
	    #sw_NumberOfFailsAux.%X0 := NOT #ix_PowerSupplyOk_1;            //  Power supply 1 state
	    #sw_NumberOfFailsAux.%X1 := NOT #ix_PowerSupplyOk_2;            //  Power supply 2 state
	    #sw_NumberOfFailsAux.%X2 := NOT #ix_PowerSupplyOk_3;            //  Power supply 3 state
	    #sw_NumberOfFailsAux.%X3 := NOT #ix_PowerSupplyOk_4;            //  Power supply 4 state
	    #sw_NumberOfFailsAux.%X4 := NOT #ix_PowerSupplyOk_5;            //  Power supply 5 state
	    #sw_NumberOfFailsAux.%X5 := NOT #ix_PowerSupplyOk_6;            //  Power supply 6 state
	    #sw_NumberOfFailsAux.%X6 := NOT #ix_PowerSupplyOk_7;            //  Power supply 7 state
	    #sw_NumberOfFailsAux.%X7 := NOT #ix_PowerSupplyOk_8;            //  Power supply 8 state
	    #sw_NumberOfFailsAux.%X8 := NOT #ix_PowerSupplyOk_9;            //  Power supply 9 state
	    #sw_NumberOfFailsAux.%X9 := NOT #ix_PowerSupplyOk_10;           //  Power supply 10 state

	    #si_NumberOfFails := BITSUM(#sw_NumberOfFailsAux);

	END_REGION

	REGION 2 - Reset

	    IF #iqUDT_EquipmentControl.Command.Reset
	    THEN

	        #sUDT_HMIStatus.Specific.Fail_PowerSupply_1 := FALSE;      //  Power supply fault state
	        #sUDT_HMIStatus.Specific.Fail_PowerSupply_2 := FALSE;      //  Power supply fault state
	        #sUDT_HMIStatus.Specific.Fail_PowerSupply_3 := FALSE;      //  Power supply fault state
	        #sUDT_HMIStatus.Specific.Fail_PowerSupply_4 := FALSE;      //  Power supply fault state
	        #sUDT_HMIStatus.Specific.Fail_PowerSupply_5 := FALSE;      //  Power supply fault state
	        #sUDT_HMIStatus.Specific.Fail_PowerSupply_6 := FALSE;      //  Power supply fault state
	        #sUDT_HMIStatus.Specific.Fail_PowerSupply_7 := FALSE;      //  Power supply fault state
	        #sUDT_HMIStatus.Specific.Fail_PowerSupply_8 := FALSE;      //  Power supply fault state
	        #sUDT_HMIStatus.Specific.Fail_PowerSupply_9 := FALSE;      //  Power supply fault state
	        #sUDT_HMIStatus.Specific.Fail_PowerSupply_10 := FALSE;     //  Power supply fault state

	        #sUDT_HMIStatus.Specific.PowerSuppliesError := FALSE;
	        #sUDT_HMIStatus.Specific.PowerSuppliesWarning := FALSE;

	    END_IF;

	END_REGION

	REGION 3 - Status

	    // Set warning if there is an error with one power supply
	    IF #si_NumberOfFails = 1
	    THEN

	        #sUDT_HMIStatus.Specific.PowerSuppliesWarning := TRUE;

	    END_IF;

	    #sx_WarningAux := (#si_NumberOfFails = 1);

	    #R_Trig_Warning(CLK := #sx_WarningAux);

	    //  Set error if there are more than one power supply with error
	    IF #si_NumberOfFails > 1
	    THEN

	        #sUDT_HMIStatus.Specific.PowerSuppliesError := TRUE;

	    END_IF;

	    #sx_ErrorAux := (#si_NumberOfFails > 1);

	    #R_Trig_Error(CLK := #sx_ErrorAux);

	    // Set error state if there is an error with the power supply 1
	    IF NOT #ix_PowerSupplyOk_1
	    THEN

	        #sUDT_HMIStatus.Specific.Fail_PowerSupply_1 := TRUE;

	    END_IF;

	    // Set error state if there is an error with the power supply 2
	    IF NOT #ix_PowerSupplyOk_2
	    THEN

	        #sUDT_HMIStatus.Specific.Fail_PowerSupply_2 := TRUE;

	    END_IF;

	    // Set error state if there is an error with the power supply 3
	    IF NOT #ix_PowerSupplyOk_3
	    THEN

	        #sUDT_HMIStatus.Specific.Fail_PowerSupply_3 := TRUE;

	    END_IF;

	    // Set error state if there is an error with the power supply 4
	    IF NOT #ix_PowerSupplyOk_4
	    THEN

	        #sUDT_HMIStatus.Specific.Fail_PowerSupply_4 := TRUE;

	    END_IF;

	    // Set error state if there is an error with the power supply 5
	    IF NOT #ix_PowerSupplyOk_5
	    THEN

	        #sUDT_HMIStatus.Specific.Fail_PowerSupply_5 := TRUE;

	    END_IF;

	    // Set error state if there is an error with the power supply 6
	    IF NOT #ix_PowerSupplyOk_6
	    THEN

	        #sUDT_HMIStatus.Specific.Fail_PowerSupply_6 := TRUE;

	    END_IF;

	    // Set error state if there is an error with the power supply 7
	    IF NOT #ix_PowerSupplyOk_7
	    THEN

	        #sUDT_HMIStatus.Specific.Fail_PowerSupply_7 := TRUE;

	    END_IF;

	    // Set error state if there is an error with the power supply 8
	    IF NOT #ix_PowerSupplyOk_8
	    THEN

	        #sUDT_HMIStatus.Specific.Fail_PowerSupply_8 := TRUE;

	    END_IF;

	    // Set error state if there is an error with the power supply 9
	    IF NOT #ix_PowerSupplyOk_9
	    THEN

	        #sUDT_HMIStatus.Specific.Fail_PowerSupply_9 := TRUE;

	    END_IF;

	    // Set error state if there is an error with the power supply 10
	    IF NOT #ix_PowerSupplyOk_10
	    THEN

	        #sUDT_HMIStatus.Specific.Fail_PowerSupply_10 := TRUE;

	    END_IF;

	END_REGION

	REGION 4 - Statistics

	    //  Warning statistics

	    IF #sx_WarningAux
	        OR #iqUDT_EquipmentControl.Command.ResetData
	    THEN

	        "FC_Statistics"(ix_Reset := #iqUDT_EquipmentControl.Command.ResetData,
	                        ix_Activate := #sUDT_HMIStatus.Specific.PowerSuppliesWarning,
	                        ix_RTrigActivate := #R_Trig_Warning.Q,
	                        iqUDT_Statistics := #iqUDT_Statistics.PowerSupplyGroupWarnning);

	    END_IF;

	    //  Error statistics

	    IF #sx_ErrorAux
	        OR #iqUDT_EquipmentControl.Command.ResetData
	    THEN

	        "FC_Statistics"(ix_Reset := #iqUDT_EquipmentControl.Command.ResetData,
	                        ix_Activate := #sUDT_HMIStatus.Specific.PowerSuppliesError,
	                        ix_RTrigActivate := #R_Trig_Error.Q,
	                        iqUDT_Statistics := #iqUDT_Statistics.PowerSupplyGroupError);

	    END_IF;

	END_REGION

	REGION 5 - Status Update

	    #sUDT_CommonStatus.Error := #sUDT_HMIStatus.Specific.PowerSuppliesError;
	    #sUDT_CommonStatus.Warning := #sUDT_HMIStatus.Specific.PowerSuppliesWarning;

	    // HMI status update
	    IF #sUDT_CommonStatusOld <> #sUDT_CommonStatus                    // update on change
	    THEN

	        // HMI status initialization
	        #sUDT_HMIStatus.Status := 0;

	        IF #sUDT_CommonStatus.Error                                    // Error
	        THEN

	            #sUDT_HMIStatus.Status := "DB_HMIStatusConfiguration".Error;

	        END_IF;

	        IF #sUDT_CommonStatus.Warning                                  // Warning
	        THEN

	            #sUDT_HMIStatus.Status := "DB_HMIStatusConfiguration".Warning;

	        END_IF;


	        #qUDT_Status := #sUDT_CommonStatus;                           // Copy status to output
	        #sUDT_CommonStatusOld := #sUDT_CommonStatus;                  // Copy status to memory

	    END_IF;
	    #qUDT_HMIStatus := #sUDT_HMIStatus;                           // Copy HMI status to output


	END_REGION

	REGION 6 - Report to control block

	    // Function to manage report between control block and equipment block

	    "FC_EquipmentReport"(iUDT_Status := #sUDT_CommonStatus,
	                         iqUDT_Control := #iqUDT_EquipmentControl);

	END_REGION

END_FUNCTION_BLOCK

FUNCTION_BLOCK "FB_InductGINControl"
{ S7_Optimized_Access := 'TRUE' }
VERSION : 0.1
// ATTRIBUTES
// AUTO_NUMBER = True
// BLOCK_NUMBER = 15
// END_ATTRIBUTES
   VAR_INPUT
      iUDT_InductConfig { ExternalAccessible := 'False'; ExternalVisible := 'False'; ExternalWritable := 'False'} : "UDT_InductConfiguration";   // Induct configuration parameters
      ii_GINAtLastPosition { ExternalAccessible := 'False'; ExternalVisible := 'False'; ExternalWritable := 'False'} : Int;   // GIN number at the last position in the FIFO
      ii_ConfirmationGIN2to1 { ExternalAccessible := 'False'; ExternalVisible := 'False'; ExternalWritable := 'False'} : Int;   // Confirmation GIN number on position 1. Is to be used to confirm the GIN number after shifting data from position 2 to position 1.
      ii_ConfirmationGIN3to2 { ExternalAccessible := 'False'; ExternalVisible := 'False'; ExternalWritable := 'False'} : Int;   // Confirmation GIN number on position 2. Is to be used to confirm the GIN number after shifting data from position 3 to position 2.
      ii_ConfirmationGIN4to3 { ExternalAccessible := 'False'; ExternalVisible := 'False'; ExternalWritable := 'False'} : Int;   // Confirmation GIN number on position 3. Is to be used to confirm the GIN number after shifting data from position 4 to position 3.
      ii_ConfirmationGIN5to4 { ExternalAccessible := 'False'; ExternalVisible := 'False'; ExternalWritable := 'False'} : Int;   // Confirmation GIN number on position 4. Is to be used to confirm the GIN number after shifting data from position 5 to position 4.
      ii_ConfirmationGIN6to5 { ExternalAccessible := 'False'; ExternalVisible := 'False'; ExternalWritable := 'False'} : Int;   // Confirmation GIN number on position 5. Is to be used to confirm the GIN number after shifting data from position 6 to position 5.
      ii_FirstShiftCheckPosition { ExternalAccessible := 'False'; ExternalVisible := 'False'; ExternalWritable := 'False'} : Int;   // First position from which shifting request is required
      ii_InductDisplacement { ExternalAccessible := 'False'; ExternalVisible := 'False'; ExternalWritable := 'False'} : Int;   // Displacement from the Induct belt, per PLC scan [cm]
      ix_TIP_Induct { ExternalAccessible := 'False'; ExternalVisible := 'False'; ExternalWritable := 'False'} : Bool;   // Transfer in progress from Induct conveyor
      ix_ConfirmationRequired1 { ExternalAccessible := 'False'; ExternalVisible := 'False'; ExternalWritable := 'False'} : Bool;   // Request for data confirmation on position 1
      ix_ConfirmationRequired2 { ExternalAccessible := 'False'; ExternalVisible := 'False'; ExternalWritable := 'False'} : Bool;   // Request for data confirmation on position 2
      ix_ConfirmationRequired3 { ExternalAccessible := 'False'; ExternalVisible := 'False'; ExternalWritable := 'False'} : Bool;   // Request for data confirmation on position 3
      ix_ConfirmationRequired4 { ExternalAccessible := 'False'; ExternalVisible := 'False'; ExternalWritable := 'False'} : Bool;   // Request for data confirmation on position 4
      ix_ConfirmationRequired5 { ExternalAccessible := 'False'; ExternalVisible := 'False'; ExternalWritable := 'False'} : Bool;   // Request for data confirmation on position 5
      ix_ShiftDataReq2to1 { ExternalAccessible := 'False'; ExternalVisible := 'False'; ExternalWritable := 'False'} : Bool;   // Request for data shifting from position 2 to position 1
      ix_ShiftDataReq3to2 { ExternalAccessible := 'False'; ExternalVisible := 'False'; ExternalWritable := 'False'} : Bool;   // Request for data shifting from position 3 to position 2
      ix_ShiftDataReq4to3 { ExternalAccessible := 'False'; ExternalVisible := 'False'; ExternalWritable := 'False'} : Bool;   // Request for data shifting from position 4 to position 3
      ix_ShiftDataReq5to4 { ExternalAccessible := 'False'; ExternalVisible := 'False'; ExternalWritable := 'False'} : Bool;   // Request for data shifting from position 5 to position 4
      ix_ShiftDataReq6to5 { ExternalAccessible := 'False'; ExternalVisible := 'False'; ExternalWritable := 'False'} : Bool;   // Request for data shifting from position 6 to position 5
      ix_EnergySaveActive { ExternalAccessible := 'False'; ExternalVisible := 'False'; ExternalWritable := 'False'} : Bool;   // Energy safe is active
      ix_ExternalError { ExternalAccessible := 'False'; ExternalVisible := 'False'; ExternalWritable := 'False'} : Bool;   // External error occure
   END_VAR

   VAR_IN_OUT
      iqUDT_Induct : "UDT_Induct";   // Induct FIFO structure
      iqUDT_MergeInterface : "UDT_ConveyorInterface";   // Interface structure of merge conveyor
      iqUDT_MergeTracking : Array[*] of Int;   // Tracking array of the merge belt
      iqUDT_HandShake : "UDT_ConveyorHandshake";   // Induct conveyor handshake structure
      iqUDT_UnknownGINRange : "UDT_UnknownGIN";   // Unknown GIN range
      iqUDT_InductStatus : "UDT_CommonStatus";   // Induct Status
   END_VAR

   VAR
      sa_ShiftData { ExternalAccessible := 'False'; ExternalVisible := 'False'; ExternalWritable := 'False'} : Array[1..#ci_Positions] of Struct   // Data shifting structure
         Request { ExternalAccessible := 'False'; ExternalVisible := 'False'; ExternalWritable := 'False'} : Bool;   // Request to shift the data
         Done { ExternalAccessible := 'False'; ExternalVisible := 'False'; ExternalWritable := 'False'} : Bool;   // Shifting is done
         OldGIN { ExternalAccessible := 'False'; ExternalVisible := 'False'; ExternalWritable := 'False'} : Int;   // Old GIN number
      END_STRUCT;
      sa_ConfirmData { ExternalAccessible := 'False'; ExternalVisible := 'False'; ExternalWritable := 'False'} : Array[1..#ci_Positions] of Struct   // Data confirmation structure
         Request { ExternalAccessible := 'False'; ExternalVisible := 'False'; ExternalWritable := 'False'} : Bool;   // Confirmation request
         Done { ExternalAccessible := 'False'; ExternalVisible := 'False'; ExternalWritable := 'False'} : Bool;   // Confirmation is done
         OldGIN { ExternalAccessible := 'False'; ExternalVisible := 'False'; ExternalWritable := 'False'} : Int;   // Old GIN number
      END_STRUCT;
      sa_Diagnostic { ExternalAccessible := 'False'; ExternalVisible := 'False'; ExternalWritable := 'False'} : Struct   // Diagnostic structure, only for commissioning purposes
         MissingWindow { ExternalAccessible := 'False'; ExternalVisible := 'False'; ExternalWritable := 'False'} : Int;
         WrongLength { ExternalAccessible := 'False'; ExternalVisible := 'False'; ExternalWritable := 'False'} : Int;
         TrackingLost { ExternalAccessible := 'False'; ExternalVisible := 'False'; ExternalWritable := 'False'} : Int;
      END_STRUCT;
      sUDT_EmptyParcelData { ExternalAccessible := 'False'; ExternalVisible := 'False'; ExternalWritable := 'False'; S7_SetPoint := 'False'} : "UDT_InductParcelData";   // Empty parcel data
      sR_Trig_ShiftDataReq2to1 {InstructionName := 'R_TRIG'; LibVersion := '1.0'; ExternalAccessible := 'False'; ExternalVisible := 'False'; ExternalWritable := 'False'; S7_SetPoint := 'False'} : R_TRIG;   // Rising edge trigger for data shifting request from position 2 to position 1
      sR_Trig_ShiftDataReq3to2 {InstructionName := 'R_TRIG'; LibVersion := '1.0'; ExternalAccessible := 'False'; ExternalVisible := 'False'; ExternalWritable := 'False'; S7_SetPoint := 'False'} : R_TRIG;   // Rising edge trigger for data shifting request from position 3 to position 2
      sR_Trig_ShiftDataReq4to3 {InstructionName := 'R_TRIG'; LibVersion := '1.0'; ExternalAccessible := 'False'; ExternalVisible := 'False'; ExternalWritable := 'False'; S7_SetPoint := 'False'} : R_TRIG;   // Rising edge trigger for data shifting request from position 4 to position 3
      sR_Trig_ShiftDataReq5to4 {InstructionName := 'R_TRIG'; LibVersion := '1.0'; ExternalAccessible := 'False'; ExternalVisible := 'False'; ExternalWritable := 'False'; S7_SetPoint := 'False'} : R_TRIG;   // Rising edge trigger for data shifting request from position 5 to position 4
      sR_Trig_ShiftDataReq6to5 {InstructionName := 'R_TRIG'; LibVersion := '1.0'; ExternalAccessible := 'False'; ExternalVisible := 'False'; ExternalWritable := 'False'; S7_SetPoint := 'False'} : R_TRIG;   // Rising edge trigger for data shifting request from position 6 to position 5
      sR_Trig_TIP {InstructionName := 'R_TRIG'; LibVersion := '1.0'; ExternalAccessible := 'False'; ExternalVisible := 'False'; ExternalWritable := 'False'; S7_SetPoint := 'False'} : R_TRIG;   // Rising edge trigger transfer in progress signal
      si_GinOld { ExternalAccessible := 'False'; ExternalVisible := 'False'; ExternalWritable := 'False'} : Int;   // Old GIN number
      si_ClearDistance { ExternalAccessible := 'False'; ExternalVisible := 'False'; ExternalWritable := 'False'} : Int;   // Distance to check if the conveyor moved after TIP is active
      si_NrOfPositions { ExternalAccessible := 'False'; ExternalVisible := 'False'; ExternalWritable := 'False'} : Int;   // Number of positions
      si_ExceptionPosition { ExternalAccessible := 'False'; ExternalVisible := 'False'; ExternalWritable := 'False'} : Int;   // Position from which is exception handling functionality started
      sx_CheclClearDistance { ExternalAccessible := 'False'; ExternalVisible := 'False'; ExternalWritable := 'False'} : Bool;   // Auxiliary variable to check if the conveyor moved after TIP is active
   END_VAR

   VAR_TEMP
      ti_LoopCounter1 : Int;   // Loop counter
      ti_LoopCounter2 : Int;   // Loop counter
   END_VAR

   VAR CONSTANT
      ci_Positions : Int := 20;   // Number of positions
      ci_RequestLengthCheckPosition : Int := 100;   // Distance from induct position when the requested length is checked [cm]
   END_VAR


BEGIN
	(*
	----------------------------------------------------------------------------------------

	Version history:
	Date        | Version   | Author        | Remark
	----------------------------------------------------------------------------------------
	23/03/2022  | 1.0       | H. Rutkowski  | First release TIA 16
	19/04/2022  | 1.1       | M. Piela      | Rebuild data shifting, add exception handling
	10/06/2022  | 1.2       | M. Piela      | When shifting data checking if the position is empty or the confirmation is not required
	22/07/2022  | 1.3       | M. Piela      | Change the condition to recover when the parcel is at the induct position but has no GIN number
	21/02/2023  | 4.0       | F.Baten       | 4.0 Release TIA 17.5
	*)

	REGION 1 - Intialize and Trigger

	    #sR_Trig_ShiftDataReq2to1(CLK := #ix_ShiftDataReq2to1);
	    #sR_Trig_ShiftDataReq3to2(CLK := #ix_ShiftDataReq3to2);
	    #sR_Trig_ShiftDataReq4to3(CLK := #ix_ShiftDataReq4to3);
	    #sR_Trig_ShiftDataReq5to4(CLK := #ix_ShiftDataReq5to4);
	    #sR_Trig_ShiftDataReq6to5(CLK := #ix_ShiftDataReq6to5);
	    #sR_Trig_TIP(CLK := #ix_TIP_Induct);

	END_REGION

	REGION 2 - Queue

	    REGION 2.1 - Position 1

	        //Clear the data on position 1 when TIP is on and the conveyor belt had moved
	        IF #sR_Trig_TIP.Q
	            AND NOT #sx_CheclClearDistance
	        THEN
	            #sx_CheclClearDistance := TRUE;
	            #si_ClearDistance := 0;
	        END_IF;

	        IF #sx_CheclClearDistance
	        THEN
	            #si_ClearDistance += #ii_InductDisplacement;
	        END_IF;

	        //Check if the conveyor belt moved after TIP occur
	        IF #si_ClearDistance > 5
	        THEN
	            #iqUDT_Induct.Position[1] := #sUDT_EmptyParcelData;
	            #sx_CheclClearDistance := FALSE;
	            #si_ClearDistance := 0;
	        END_IF;

	    END_REGION

	    REGION 2.2 - Position 2 to 1

	        //Shift Data
	        IF #sR_Trig_ShiftDataReq2to1.Q // External request for shifting data
	        THEN
	            #sa_ShiftData[2].Request := TRUE; // Request data shifting
	            #sa_ShiftData[2].Done := FALSE;   // Set shift data done to false
	        END_IF;

	        IF (#sa_ShiftData[2].Request
	            OR #ii_FirstShiftCheckPosition < 1)     // Check if the check position is less than the position from which shifting request is required
	            AND (#iqUDT_Induct.Position[2].GINNumber > 0 AND #iqUDT_Induct.Position[1].GINNumber = 0)  //Check if the data to be moved are present and the position the data will be moved to is empty
	            AND ((#sa_ConfirmData[2].Done AND #ix_ConfirmationRequired2) OR NOT #ix_ConfirmationRequired2)    //Validate if the data were confirmed if confirmation configured
	        THEN
	            #iqUDT_Induct.Position[1] := #iqUDT_Induct.Position[2]; //Shift the data
	            #iqUDT_Induct.Position[2] := #sUDT_EmptyParcelData;    //Clear the data on the position from where the data were shifted
	            #sa_ShiftData[2].Request := FALSE;
	            #sa_ShiftData[2].Done := TRUE;
	            #sa_ConfirmData[1].Request := #ix_ConfirmationRequired1; // Request data confirmation if configured
	            #sa_ConfirmData[1].Done := FALSE;
	        END_IF;

	        // Confirm data
	        IF #sa_ConfirmData[1].Request
	            AND #ii_ConfirmationGIN2to1 <> 0
	            AND #iqUDT_Induct.Position[1].GINNumber > 0
	            AND #sa_ConfirmData[1].OldGIN <> #ii_ConfirmationGIN2to1   //Check if confirmation GIN is different than the old confirmation GIN
	            AND #ii_ConfirmationGIN2to1 <> #ii_ConfirmationGIN3to2    //Check if confirmation GIN is different than confirmation GIN in previous position
	        THEN
	            IF #iqUDT_Induct.Position[1].GINNumber = #ii_ConfirmationGIN2to1 //Validate if the GIN number matches the GIN number on the confirmation position
	            THEN
	                #sa_ConfirmData[1].Done := TRUE;
	                #sa_ConfirmData[1].Request := FALSE;
	                #sa_ConfirmData[1].OldGIN := #ii_ConfirmationGIN2to1;

	            ELSE
	                // Data lost, overwrite with confirmation data
	                #iqUDT_Induct.Position[1] := #sUDT_EmptyParcelData;
	                #iqUDT_Induct.Position[1].GINNumber := #ii_ConfirmationGIN2to1;

	                //Write maximum requested gap
	                #iqUDT_Induct.Position[1].GapRequired := (#iUDT_InductConfig.MaxParcelSize / 10) + #iUDT_InductConfig.GapTailToHead;

	                #sa_ConfirmData[1].OldGIN := #ii_ConfirmationGIN2to1;
	                #sa_ConfirmData[1].Done := TRUE;
	                #sa_ConfirmData[1].Request := FALSE;
	                #si_ExceptionPosition := 1; //Write exception position the same as a position on which data were lost
	            END_IF;

	        END_IF;

	    END_REGION

	    REGION 2.3 - Position 3 to 2

	        IF #sR_Trig_ShiftDataReq3to2.Q // External request for shifting data
	        THEN

	            #sa_ShiftData[3].Request := TRUE; // Request data shifting
	            #sa_ShiftData[3].Done := FALSE;   // Set shift data done to false

	        END_IF;

	        IF (#sa_ShiftData[3].Request
	            OR #ii_FirstShiftCheckPosition < 2)         // Check if the check position is less than the position from which shifting request is required
	            AND (#iqUDT_Induct.Position[3].GINNumber > 0 AND (#iqUDT_Induct.Position[2].GINNumber = 0 OR NOT #ix_ConfirmationRequired2)) //Check if the data to be moved are present and the position the data will be moved to is empty
	            AND ((#sa_ConfirmData[3].Done AND #ix_ConfirmationRequired3) OR NOT #ix_ConfirmationRequired3)    //Validate if the data were confirmed if confirmation configured
	        THEN
	            #iqUDT_Induct.Position[2] := #iqUDT_Induct.Position[3]; //Shift the data
	            #iqUDT_Induct.Position[3] := #sUDT_EmptyParcelData;     //Clear the data on the position from where the data were shifted
	            #sa_ShiftData[3].Request := FALSE;
	            #sa_ShiftData[3].Done := TRUE;
	            #sa_ConfirmData[2].Request := #ix_ConfirmationRequired2;   // Request data confirmation if configured
	            #sa_ConfirmData[2].Done := FALSE;
	        END_IF;

	        //Cofirm data
	        IF #sa_ConfirmData[2].Request
	            AND #ii_ConfirmationGIN3to2 <> 0
	            AND #iqUDT_Induct.Position[2].GINNumber > 0
	            AND #sa_ConfirmData[2].OldGIN <> #ii_ConfirmationGIN3to2 //Check if confirmation GIN is different than the old confirmation GIN
	            AND #ii_ConfirmationGIN4to3 <> #ii_ConfirmationGIN3to2  //Check if confirmation GIN is different than confirmation GIN in previous position
	        THEN

	            IF #iqUDT_Induct.Position[2].GINNumber = #ii_ConfirmationGIN3to2  //Validate if the GIN number matches the GIN number on the confirmation position

	            THEN
	                #sa_ConfirmData[2].Done := TRUE;
	                #sa_ConfirmData[2].Request := FALSE;
	                #sa_ConfirmData[2].OldGIN := #ii_ConfirmationGIN3to2;

	            ELSE
	                // Data lost, overwrite with confirmation data
	                #iqUDT_Induct.Position[2] := #sUDT_EmptyParcelData;
	                #iqUDT_Induct.Position[2].GINNumber := #ii_ConfirmationGIN3to2;

	                //Write maximum requested gap
	                #iqUDT_Induct.Position[2].GapRequired := (#iUDT_InductConfig.MaxParcelSize / 10) + #iUDT_InductConfig.GapTailToHead;

	                #sa_ConfirmData[2].OldGIN := #ii_ConfirmationGIN3to2;
	                #sa_ConfirmData[2].Done := TRUE;
	                #sa_ConfirmData[2].Request := FALSE;
	                #si_ExceptionPosition := 2; //Write exception position the same as a position on which data were lost
	            END_IF;

	        END_IF;

	    END_REGION

	    REGION 2.4 - Position 4 to 3

	        IF #sR_Trig_ShiftDataReq4to3.Q // External request for shifting data
	        THEN

	            #sa_ShiftData[4].Request := TRUE; // Request data shifting
	            #sa_ShiftData[4].Done := FALSE;   // Set shift data done to false
	        END_IF;

	        IF (#sa_ShiftData[4].Request
	            OR #ii_FirstShiftCheckPosition < 3)     // Check if the check position is less than the position from which shifting request is required
	            AND (#iqUDT_Induct.Position[4].GINNumber > 0 AND (#iqUDT_Induct.Position[3].GINNumber = 0 OR NOT #ix_ConfirmationRequired3)) //Check if the data to be moved are present and the position the data will be moved to is empty.
	            AND ((#sa_ConfirmData[4].Done AND #ix_ConfirmationRequired4) OR NOT #ix_ConfirmationRequired4)    //Validate if the data were confirmed if confirmation configured
	        THEN
	            #iqUDT_Induct.Position[3] := #iqUDT_Induct.Position[4]; //Shift the data
	            #iqUDT_Induct.Position[4] := #sUDT_EmptyParcelData;     //Clear the data on the position from where the data were shifted
	            #sa_ShiftData[4].Request := FALSE;
	            #sa_ShiftData[4].Done := TRUE;
	            #sa_ConfirmData[3].Request := #ix_ConfirmationRequired3;   // Request data confirmation if configured
	            #sa_ConfirmData[3].Done := FALSE;
	        END_IF;

	        // Confirm data
	        IF #sa_ConfirmData[3].Request
	            AND #ii_ConfirmationGIN4to3 <> 0
	            AND #iqUDT_Induct.Position[3].GINNumber > 0
	            AND #sa_ConfirmData[3].OldGIN <> #ii_ConfirmationGIN4to3 //Check if confirmation GIN is different than the old confirmation GIN
	            AND #ii_ConfirmationGIN4to3 <> #ii_ConfirmationGIN5to4  //Check if confirmation GIN is different than confirmation GIN in previous position

	        THEN
	            IF #iqUDT_Induct.Position[3].GINNumber = #ii_ConfirmationGIN4to3  //Validate if the GIN number matches the GIN number on the confirmation position
	            THEN
	                #sa_ConfirmData[3].Done := TRUE;
	                #sa_ConfirmData[3].Request := FALSE;
	                #sa_ConfirmData[3].OldGIN := #ii_ConfirmationGIN4to3;
	            ELSE
	                // Data lost, overwrite with confirmation data
	                #iqUDT_Induct.Position[3] := #sUDT_EmptyParcelData;
	                #iqUDT_Induct.Position[3].GINNumber := #ii_ConfirmationGIN4to3;

	                //Write maximum requested gap
	                #iqUDT_Induct.Position[3].GapRequired := (#iUDT_InductConfig.MaxParcelSize / 10) + #iUDT_InductConfig.GapTailToHead;

	                #sa_ConfirmData[3].OldGIN := #ii_ConfirmationGIN4to3;
	                #sa_ConfirmData[3].Done := TRUE;
	                #sa_ConfirmData[3].Request := FALSE;
	                #si_ExceptionPosition := 3; //Write exception position the same as a position on which data were lost
	            END_IF;

	        END_IF;

	    END_REGION

	    REGION 2.5 - Position 5 to 4

	        IF #sR_Trig_ShiftDataReq5to4.Q // External request for shifting data
	        THEN

	            #sa_ShiftData[5].Request := TRUE; // Request data shifting
	            #sa_ShiftData[5].Done := FALSE;   // Set shift data done to false

	        END_IF;

	        IF (#sa_ShiftData[5].Request
	            OR #ii_FirstShiftCheckPosition < 4)     // Check if the check position is less than the position from which shifting request is required
	            AND (#iqUDT_Induct.Position[5].GINNumber > 0 AND (#iqUDT_Induct.Position[4].GINNumber = 0 OR NOT #ix_ConfirmationRequired4)) //Check if the data to be moved are present and the position the data will be moved to is empty.
	            AND ((#sa_ConfirmData[5].Done AND #ix_ConfirmationRequired5) OR NOT #ix_ConfirmationRequired5) //Validate if the data were confirmed if confirmation configured
	        THEN
	            #iqUDT_Induct.Position[4] := #iqUDT_Induct.Position[5]; //Shift the data
	            #iqUDT_Induct.Position[5] := #sUDT_EmptyParcelData;    //Clear the data on the position from where the data were shifted
	            #sa_ShiftData[5].Request := FALSE;
	            #sa_ShiftData[5].Done := TRUE;
	            #sa_ConfirmData[4].Request := #ix_ConfirmationRequired4;   // Request data confirmation if configured
	            #sa_ConfirmData[4].Done := FALSE;
	        END_IF;

	        // Confirm data
	        IF #sa_ConfirmData[4].Request
	            AND #ii_ConfirmationGIN5to4 <> 0
	            AND #iqUDT_Induct.Position[4].GINNumber > 0
	            AND #sa_ConfirmData[4].OldGIN <> #ii_ConfirmationGIN5to4 //Check if confirmation GIN is different than the old confirmation GIN
	            AND #ii_ConfirmationGIN5to4 <> #ii_ConfirmationGIN6to5  //Check IF confirmation GIN is different than confirmation GIN in previous position
	        THEN
	            IF #iqUDT_Induct.Position[4].GINNumber = #ii_ConfirmationGIN5to4  //Validate if the GIN number matches the GIN number on the confirmation position
	            THEN
	                #sa_ConfirmData[4].Done := TRUE;
	                #sa_ConfirmData[4].Request := FALSE;
	                #sa_ConfirmData[4].OldGIN := #ii_ConfirmationGIN5to4;
	            ELSE
	                // Data lost, overwrite with confirmation data
	                #iqUDT_Induct.Position[4] := #sUDT_EmptyParcelData;
	                #iqUDT_Induct.Position[4].GINNumber := #ii_ConfirmationGIN5to4;

	                //Write maximum requested gap
	                #iqUDT_Induct.Position[4].GapRequired := (#iUDT_InductConfig.MaxParcelSize / 10) + #iUDT_InductConfig.GapTailToHead;

	                #sa_ConfirmData[4].OldGIN := #ii_ConfirmationGIN5to4;
	                #sa_ConfirmData[4].Done := TRUE;
	                #sa_ConfirmData[4].Request := FALSE;
	                #si_ExceptionPosition := 4; //Write exception position the same as a position on which data were lost
	            END_IF;
	        END_IF;

	    END_REGION

	    REGION 2.6 - Position 6 to 5


	        IF #sR_Trig_ShiftDataReq6to5.Q // External request for shifting data
	        THEN

	            #sa_ShiftData[6].Request := TRUE; // Request data shifting
	            #sa_ShiftData[6].Done := FALSE;   // Set shift data done to false

	        END_IF;

	        IF (#sa_ShiftData[6].Request
	            OR #ii_FirstShiftCheckPosition < 5)     // Check if the check position is less than the position from which shifting request is required
	            AND (#iqUDT_Induct.Position[6].GINNumber > 0 AND (#iqUDT_Induct.Position[5].GINNumber = 0 OR NOT #ix_ConfirmationRequired5)) //Check if the data to be moved are present and the position the data will be moved to is empty.
	        THEN
	            #iqUDT_Induct.Position[5] := #iqUDT_Induct.Position[6]; //Shift the data
	            #iqUDT_Induct.Position[6] := #sUDT_EmptyParcelData;     //Clear the data on the position from where the data were shifted
	            #sa_ShiftData[6].Request := FALSE;
	            #sa_ShiftData[6].Done := TRUE;
	            #sa_ConfirmData[5].Request := #ix_ConfirmationRequired5; // Request data confirmation if configured
	            #sa_ConfirmData[5].Done := FALSE;
	        END_IF;

	        // Confirm data
	        IF #sa_ConfirmData[5].Request
	            AND #ii_ConfirmationGIN6to5 <> 0
	            AND #iqUDT_Induct.Position[5].GINNumber > 0
	            AND #sa_ConfirmData[5].OldGIN <> #ii_ConfirmationGIN6to5 //Check if confirmation GIN is different than the old confirmation GIN
	        THEN
	            IF #iqUDT_Induct.Position[5].GINNumber = #ii_ConfirmationGIN6to5 //Validate if the GIN number matches the GIN number on the confirmation position
	            THEN
	                #sa_ConfirmData[5].Done := TRUE;
	                #sa_ConfirmData[5].Request := FALSE;
	                #sa_ConfirmData[5].OldGIN := #ii_ConfirmationGIN6to5;
	            ELSE
	                // Data lost, overwrite with confirmation data
	                #iqUDT_Induct.Position[5] := #sUDT_EmptyParcelData;
	                #iqUDT_Induct.Position[5].GINNumber := #ii_ConfirmationGIN6to5;

	                //Write maximum requested gap
	                #iqUDT_Induct.Position[5].GapRequired := (#iUDT_InductConfig.MaxParcelSize / 10) + #iUDT_InductConfig.GapTailToHead;

	                #sa_ConfirmData[5].OldGIN := #ii_ConfirmationGIN6to5;
	                #sa_ConfirmData[5].Done := TRUE;
	                #sa_ConfirmData[5].Request := FALSE;
	                #si_ExceptionPosition := 5;    //Write exception position the same as a position on which data were lost
	            END_IF;
	        END_IF;

	    END_REGION

	    REGION 2.7 - Adding new parcel to the induct

	        // Check if the GIN number at the last position if grather than 0
	        IF #ii_GINAtLastPosition > 0
	            AND #ii_GINAtLastPosition <> #si_GinOld // Check if the GIN number is different than OLD GIN
	        THEN
	            #iqUDT_Induct.Position[6].GINNumber := #ii_GINAtLastPosition;

	            IF "DB_GIN".GIN[#ii_GINAtLastPosition].General.Length > 0  //Check if the package length for the GIN number is greater than 0
	            THEN
	                #iqUDT_Induct.Position[6].GapRequired := "DB_GIN".GIN[#ii_GINAtLastPosition].General.Length + #iUDT_InductConfig.GapTailToHead; //Required gap is parcel length + configured gap tail to head
	            ELSE
	                #iqUDT_Induct.Position[6].GapRequired := (#iUDT_InductConfig.MaxParcelSize / 10) + #iUDT_InductConfig.GapTailToHead;  //Write maximum requested gap
	            END_IF;

	            #si_GinOld := #ii_GINAtLastPosition;
	        END_IF;

	    END_REGION

	    // Update diagnostic
	    IF #si_ExceptionPosition > 0
	    THEN

	        #sa_Diagnostic.TrackingLost += 1;
	    END_IF;

	END_REGION

	REGION 3 - Exceptions

	    REGION 3.1 - Window monitoring

	        //Get the number of array elements
	        #si_NrOfPositions := "FC_GetNrOfArrayEl"(#iqUDT_Induct.Position);

	        //Lookig for the missing window
	        FOR #ti_LoopCounter1 := 1 TO #si_NrOfPositions DO

	            IF #iqUDT_Induct.Position[#ti_LoopCounter1].WindowReserved //Check if window is reserved for induct position
	            THEN
	                //When the window was reserved then decrease the window position based on displacement
	                #iqUDT_Induct.Position[#ti_LoopCounter1].WindowPosition -= #iqUDT_MergeInterface.Displacement;

	                // Check if the window position value does not go negative
	                IF #iqUDT_Induct.Position[#ti_LoopCounter1].WindowPosition < 0
	                THEN
	                    #iqUDT_Induct.Position[#ti_LoopCounter1].WindowPosition := 0;
	                END_IF;
	                //When the window position is less than the induct position it means that the induct miss the window
	                IF #iqUDT_Induct.Position[#ti_LoopCounter1].WindowPosition < (#iUDT_InductConfig.Induct_Position / 10 - #iUDT_InductConfig.InductPositionWindow)
	                THEN
	                    //Write exception position
	                    IF #si_ExceptionPosition > #ti_LoopCounter1 OR #si_ExceptionPosition = 0
	                    THEN
	                        #sa_Diagnostic.MissingWindow += 1;
	                        #si_ExceptionPosition := #ti_LoopCounter1;
	                    END_IF;

	                    EXIT;
	                END_IF;

	            END_IF;

	        END_FOR;

	    END_REGION

	    REGION 3.2 - Requested length check

	        // Checking if the requested length is the same on induct array and reserved in the merge tracking array
	        FOR #ti_LoopCounter2 := ((#iUDT_InductConfig.Induct_Position / 10) + #ci_RequestLengthCheckPosition) TO ((#iUDT_InductConfig.Induct_Position / 10) + #ci_RequestLengthCheckPosition) + 5 DO
	            //When we find request to release in merge tracking array then we can check the requested length and GIN number
	            IF #iqUDT_MergeTracking[#ti_LoopCounter2] = - (#iUDT_InductConfig.Induct_Number + 100) AND
	                (#iqUDT_MergeTracking[#ti_LoopCounter2 + 1] <> #iqUDT_Induct.Position[1].GapRequired)
	                // OR #iq_UDT_MergeTracking[#ti_LoopCounter2 + 2] <> #iq_UDT_Induct.Position[1].GINNumber)
	            THEN
	                //When the requested length is different than the length reserved in the merge tracking array then we reset that request because is not valid
	                #iqUDT_MergeTracking[#ti_LoopCounter2] := 0;
	                #iqUDT_MergeTracking[#ti_LoopCounter2 + 1] := 0;
	                #iqUDT_MergeTracking[#ti_LoopCounter2 + 2] := 0;

	                #sa_Diagnostic.WrongLength += 1;

	                //Write exception position
	                IF #si_ExceptionPosition > 2 OR #si_ExceptionPosition = 0
	                THEN
	                    #si_ExceptionPosition := 1;
	                END_IF;

	                EXIT;
	            END_IF;
	        END_FOR;

	    END_REGION

	    REGION 3.3 - Lack of GIN number, auto recovey

	        // Check if the unknown GIN is within range
	        IF #iqUDT_UnknownGINRange.GIN < #iqUDT_UnknownGINRange.Start
	            OR #iqUDT_UnknownGINRange.GIN > #iqUDT_UnknownGINRange.End
	        THEN
	            #iqUDT_UnknownGINRange.GIN := #iqUDT_UnknownGINRange.Start;
	        END_IF;

	        //When the parcel is at the induct position but has no GIN number
	        IF ((#iqUDT_HandShake.RTS OR #iqUDT_InductStatus.Dieback)
	            AND #iqUDT_InductStatus.AutoON
	            AND (#iqUDT_Induct.Position[1].GINNumber = 0))

	            // Auto recovey signal from induct
	            OR #iqUDT_Induct.AutoRecovery

	        THEN
	            #si_ExceptionPosition := 1;
	            #iqUDT_Induct.Position[1].GINNumber := #iqUDT_UnknownGINRange.GIN;  //Write GIN number from Unknown GIN range
	            #iqUDT_UnknownGINRange.GIN := #iqUDT_UnknownGINRange.GIN + 1; // Update Unknown GIN range
	            #iqUDT_Induct.Position[1].GapRequired := (#iUDT_InductConfig.MaxParcelSize / 10) + #iUDT_InductConfig.GapTailToHead; //Write maximum required gap

	        END_IF;

	    END_REGION

	    REGION 3.4 - Exception handling

	        //When the exception was found reinitialize the whole array from the exception position
	        IF #si_ExceptionPosition > 0
	        THEN

	            FOR #ti_LoopCounter1 := #si_ExceptionPosition TO #si_NrOfPositions DO

	                IF #iqUDT_Induct.Position[#ti_LoopCounter1].WindowReserved //Check if window is reserved for induct position
	                THEN
	                    FOR #ti_LoopCounter2 := #iqUDT_Induct.Position[#ti_LoopCounter1].WindowPosition - 2 TO #iqUDT_Induct.Position[#ti_LoopCounter1].WindowPosition + 2 DO
	                        IF #iqUDT_MergeTracking[#ti_LoopCounter2] = - (#iUDT_InductConfig.Induct_Number + 100)
	                        THEN
	                            //Delete induct request and induct requested length
	                            #iqUDT_MergeTracking[#ti_LoopCounter2] := 0;
	                            #iqUDT_MergeTracking[#ti_LoopCounter2 + 1] := 0;
	                            #iqUDT_MergeTracking[#ti_LoopCounter2 + 2] := 0;
	                        END_IF;
	                    END_FOR;
	                    //Reset the window
	                    #iqUDT_Induct.Position[#ti_LoopCounter1].WindowPosition := 0;
	                    #iqUDT_Induct.Position[#ti_LoopCounter1].WindowReserved := FALSE;
	                ELSE
	                    EXIT;
	                END_IF;

	            END_FOR;

	        END_IF;
	        //Reset the Exception position
	        #si_ExceptionPosition := 0;

	    END_REGION

	    REGION 3.5 - Data clearing

	        //Clear remaining data when energy save occur
	        IF #ix_EnergySaveActive
	        THEN
	            FOR #ti_LoopCounter1 := 1 TO #si_NrOfPositions DO
	                #iqUDT_Induct.Position[#ti_LoopCounter1] := #sUDT_EmptyParcelData;
	            END_FOR;
	        END_IF;

	        //Disable window reservation when external error occur
	        #iqUDT_Induct.DisableWindowReservation := #ix_ExternalError;

	    END_REGION

	    REGION 3.6 - Confirm no duplicate GIN in FIFO

	        //Check FIFO in case of duplicate GIN number
	        FOR #ti_LoopCounter1 := 1 TO #si_NrOfPositions - 1 DO
	            FOR #ti_LoopCounter2 := #ti_LoopCounter1 + 1 TO #si_NrOfPositions - 1 DO
	                // When duplicate GIN number is find then clear the duplicate data
	                IF #iqUDT_Induct.Position[#ti_LoopCounter1].GINNumber = #iqUDT_Induct.Position[#ti_LoopCounter2].GINNumber
	                    AND #iqUDT_Induct.Position[#ti_LoopCounter2].GINNumber <> 0
	                THEN
	                    #iqUDT_Induct.Position[#ti_LoopCounter2] := #sUDT_EmptyParcelData;

	                END_IF;
	            END_FOR;

	        END_FOR;

	    END_REGION

	END_REGION
END_FUNCTION_BLOCK

FUNCTION_BLOCK "FB_GetGIN"
TITLE = FB_GetGIN
{ S7_Optimized_Access := 'TRUE' }
AUTHOR : MHSE
FAMILY : GeneralSystemFunctions
VERSION : 3.0
// ATTRIBUTES
// AUTO_NUMBER = True
// BLOCK_NUMBER = 10
// END_ATTRIBUTES
//Function block to find GIN in tracking array.
   VAR_INPUT
      ii_TriggerPosition { ExternalAccessible := 'False'; ExternalVisible := 'False'; ExternalWritable := 'False'} : Int;   // Position of trigger [cm]
      ii_SearchWindow { ExternalAccessible := 'False'; ExternalVisible := 'False'; ExternalWritable := 'False'} : Int;   // Search window [cm]
      ix_Trigger { ExternalAccessible := 'False'; ExternalVisible := 'False'; ExternalWritable := 'False'} : Bool;   // When TRUE get GIN code
   END_VAR

   VAR_OUTPUT
      qi_Gin { ExternalAccessible := 'False'; ExternalVisible := 'False'; ExternalWritable := 'False'} : Int;   // General Identification Number found
   END_VAR

   VAR_IN_OUT
      iqa_TrackingData : Array[*] of Int;   // Tracking data
      iqx_Received { ExternalAccessible := 'False'; ExternalVisible := 'False'; ExternalWritable := 'False'} : Bool;   // When TRUE qi_GIN output is set to '0'
   END_VAR

   VAR
      sR_Trigger {InstructionName := 'R_TRIG'; LibVersion := '1.0'; ExternalAccessible := 'False'; ExternalVisible := 'False'; ExternalWritable := 'False'; S7_SetPoint := 'False'} : R_TRIG;
      si_Loopcounter { ExternalAccessible := 'False'; ExternalVisible := 'False'; ExternalWritable := 'False'} : Int;
      si_Position { ExternalAccessible := 'False'; ExternalVisible := 'False'; ExternalWritable := 'False'} : Int;   // Position to look for Gin
      si_PosFound { ExternalAccessible := 'False'; ExternalVisible := 'False'; ExternalWritable := 'False'} : Int;   // Position first Gin was found
      sx_Found { ExternalAccessible := 'False'; ExternalVisible := 'False'; ExternalWritable := 'False'} : Bool;
   END_VAR


BEGIN
	(*
	----------------------------------------------------------------------------------------

	Version history:
	Date        | Version   | Author        | Remark
	----------------------------------------------------------------------------------------
	28/05/2019  | 0.1       | F.Baten       | first release TIA 15
	24/07/2019  | 2.0       | L.Klar        | 2.0 MHS library release TIA 15.1
	12/11/2019  | 3.0       | P.Majka       | 3.0 MHS library release TIA 15.1
	21/02/2023  | 4.0       | F.Baten       | 4.0 Release TIA 17.5


	                               Trigger
	XXX                            position                                       0
	|                                  |                                          |
	|-----------------------------------------------------------------------------|
	|                   |              |                                          |
	|                    <---window--->                               >-- tracking/flow direction -->
	|                                                                             |
	|-----------------------------------------------------------------------------|

	At a trigger pulse a Gin-code is searched in the tracking DB starting from the trigger position.
	When found the block provides the found GIN and the position it was found on.

	When the Gin was handled it can also reset the found value to 0.
	*)

	REGION 1 Get GIN from tracking DB
	    #sR_Trigger(CLK := #ix_Trigger);

	    IF #sR_Trigger.Q                                                                    // One shot to start searching in tracking DB
	    THEN
	        #qi_Gin := 0;                                                                   // reset GIN found
	        #si_Position := 0;                                                              // reset position found
	        #sx_Found := FALSE;                                                             // reset found bit


	        FOR #si_Loopcounter := 0 TO #ii_SearchWindow BY 1 DO                            // Set loopsize by search window

	            #si_Position := #ii_TriggerPosition + #si_Loopcounter;                      // Set position to look for GIN

	            IF #iqa_TrackingData[#si_Position] <> 0 AND #sx_Found = FALSE THEN          // If there is a value within the search window
	                #si_PosFound := #si_Position;
	                #qi_Gin := #iqa_TrackingData[#si_Position];                             // copy that value to output
	                #sx_Found := TRUE;                                                      // Set found
	                EXIT;
	                // EXIT loop
	            END_IF;
	        END_FOR;
	    END_IF;
	END_REGION

	REGION 2 Reset GIN, was handled
	    IF #iqx_Received                                                                    // External signal meaning GIN was received and handled
	    THEN
	        #qi_Gin := 0;                                                                   // Reset output
	        #sx_Found := FALSE;                                                             // Reset found signal
	        #iqx_Received := FALSE;                                                         // Reset handshake
	    END_IF;
	END_REGION

END_FUNCTION_BLOCK

FUNCTION_BLOCK "FB_GetPositionBasic"
TITLE = FB_GetPosition
{ S7_Optimized_Access := 'TRUE' }
FAMILY : MHS
VERSION : 3.0
// ATTRIBUTES
// AUTO_NUMBER = True
// BLOCK_NUMBER = 11
// END_ATTRIBUTES
//Function to find the position based on the GIN in the tracking.
   VAR_INPUT
      ii_Decisionpoint { ExternalAccessible := 'False'; ExternalVisible := 'False'; ExternalWritable := 'False'} : Int;   // Point in tracking data to look for GIN
   END_VAR

   VAR_IN_OUT
      iqs_DB_Destination : Array[*] of "UDT_Destinations";   // Array with destination data for parcel
      iqs_TrackingData : Array[*] of Int;   // Tracking data
      iqi_RequestedPosition { ExternalAccessible := 'False'; ExternalVisible := 'False'; ExternalWritable := 'False'} : Int;   // Requested position to go to based on GIN
   END_VAR

   VAR
      sdi_RequestedDestination { ExternalAccessible := 'False'; ExternalVisible := 'False'; ExternalWritable := 'False'} : DInt;   // The destination for this GIN
      si_Gin { ExternalAccessible := 'False'; ExternalVisible := 'False'; ExternalWritable := 'False'} : Int;   // GIN found in tracking
      si_PreviousGin { ExternalAccessible := 'False'; ExternalVisible := 'False'; ExternalWritable := 'False'} : Int;   // Previous GIN processed
      si_RequestedPosition { ExternalAccessible := 'False'; ExternalVisible := 'False'; ExternalWritable := 'False'} : Int;   // Requested position to go to based on GIN
      si_LC_Positions { ExternalAccessible := 'False'; ExternalVisible := 'False'; ExternalWritable := 'False'} : Int;   // Loopcounter positions
      si_LC_Destinations { ExternalAccessible := 'False'; ExternalVisible := 'False'; ExternalWritable := 'False'} : Int;   // Loopcounter destinations
      si_NrPositons { ExternalAccessible := 'False'; ExternalVisible := 'False'; ExternalWritable := 'False'} : Int;   // Number of positions in the search area
      si_NrDestinations { ExternalAccessible := 'False'; ExternalVisible := 'False'; ExternalWritable := 'False'} : Int;   // Number of destinations per position
      sx_NewGinFound { ExternalAccessible := 'False'; ExternalVisible := 'False'; ExternalWritable := 'False'} : Bool;   // Memory to start searching
   END_VAR


BEGIN
	(*
	----------------------------------------------------------------------------------------

	Version history:
	Date        | Version   | Author        | Remark
	----------------------------------------------------------------------------------------

	10-09-2019  | 2.0       | F.Baten       | Doubled search loop and added comment
	12/11/2019  | 3.0       | P.Majka       | 3.0 MHS library release TIA 15.1
	08/01/2020  | 3.1       | F.Baten       | When no destination is given, also go to default direction
	15/01/2019  | 3.2       | L.Klar        | GIN record structure updated, parcel destination remapped
	19/10/2020  | 3.3       | L.Klar        | Double search loop reprogrammed, issue with default position
	07/12/2020  | 3.4       | L.Klar        | GIN greater than zero condition added to region 2
	11/04/2023  | 4.0       | F.Baten       | Removed VSU interface to be adaptable for more devices
	                                        | 4.0 Release TIA 17.5
	12/
	*)


	REGION 1 - Determine size OF search area

	    #si_NrPositons := "FC_GetNrOfArrayEl"(#iqs_DB_Destination);
	    #si_NrDestinations := "FC_GetNrOfArrayEl"(#iqs_DB_Destination[1].Destination);

	END_REGION

	REGION 2 - Get GIN from tracking DB
	    // There is a value in the tracking data on the decision point which is not '0' or equal to the previous GIN

	    IF (#iqs_TrackingData[#ii_Decisionpoint] <> 0) AND (#iqs_TrackingData[#ii_Decisionpoint] <> #si_PreviousGin)
	    THEN
	        #si_Gin := #iqs_TrackingData[#ii_Decisionpoint];
	        #sx_NewGinFound := TRUE;
	    END_IF;

	END_REGION

	REGION 2 - Get destination from GIN DB
	    // If new GIN has been detected, get destination from its GIN record

	    IF #sx_NewGinFound AND #si_Gin > 0
	    THEN
	        #sdi_RequestedDestination := "DB_GIN".GIN[#si_Gin].General.Destination[0];
	        #si_PreviousGin := #si_Gin;
	        #si_Gin := 0;
	        #iqi_RequestedPosition := 0;
	    END_IF;

	END_REGION

	REGION 3 - Get requested position when new GIN is found
	    IF #sx_NewGinFound
	    THEN
	        // If destination is different than 0, find a position in destination arrays. Otherwise, requested position is set to default.
	        IF #sdi_RequestedDestination <> 0 THEN
	            FOR #si_LC_Positions := 1 TO #si_NrPositons BY 1 DO
	                FOR #si_LC_Destinations := 0 TO (#si_NrDestinations - 1) BY 1 DO
	                    IF #iqs_DB_Destination[#si_LC_Positions].Destination[#si_LC_Destinations] = #sdi_RequestedDestination
	                    THEN
	                        #si_RequestedPosition := #si_LC_Positions;
	                        EXIT;
	                    END_IF;
	                END_FOR;
	                // Position found
	                IF #si_RequestedPosition <> 0
	                THEN
	                    #iqi_RequestedPosition := #si_RequestedPosition;
	                    #sx_NewGinFound := FALSE;
	                    #si_RequestedPosition := 0;
	                    EXIT;
	                END_IF;
	            END_FOR;
	        ELSE
	            // Default position
	            #iqi_RequestedPosition := 99;
	            #sx_NewGinFound := FALSE;
	            #si_RequestedPosition := 0;
	        END_IF;
	    END_IF;
	END_REGION
END_FUNCTION_BLOCK

FUNCTION "FC_ExtractCodeFromString" : Void
{ S7_Optimized_Access := 'TRUE' }
VERSION : 0.1
   VAR_INPUT
      is_String : String;
   END_VAR

   VAR_OUTPUT
      qs_String : String;
   END_VAR

   VAR_TEMP
      ts_String : Bool;
      ti_StartPoint : Int;
      ti_StopPoint : Int;
      ti_CodeLenght : Int;
   END_VAR

   VAR CONSTANT
      StartSign : String := '$02';
      StopSign : String := '$03';
   END_VAR


BEGIN
	#ti_StartPoint := FIND(IN1 := #is_String, IN2 := #StartSign);
	#ti_StopPoint := FIND(IN1 := #is_String, IN2 := #StopSign);
	#ti_CodeLenght := #ti_StopPoint - #ti_StartPoint - 1;

	#qs_String := MID(IN := #is_String, L := #ti_CodeLenght, P := #ti_StartPoint + 1);

END_FUNCTION

FUNCTION_BLOCK "FB_GetPositionVSU"
TITLE = FB_GetPosition
{ S7_Optimized_Access := 'TRUE' }
FAMILY : MHS
VERSION : 3.0
// ATTRIBUTES
// AUTO_NUMBER = True
// BLOCK_NUMBER = 12
// END_ATTRIBUTES
//Function to find the position based on the GIN in the tracking.
   VAR_IN_OUT
      iqa_DBDestination : Array[*] of "UDT_Destinations";   // Array with destination data for parcel
      iqUDT_VSUInterface : "UDT_VSUInterface";   // Interface beween VSU and VFD
      iqa_TrackingData : Array[*] of Int;   // Tracking data
   END_VAR

   VAR
      sdi_RequestedDestination { ExternalAccessible := 'False'; ExternalVisible := 'False'; ExternalWritable := 'False'} : DInt;   // The destination for this GIN
      si_Gin { ExternalAccessible := 'False'; ExternalVisible := 'False'; ExternalWritable := 'False'} : Int;
      si_PreviousGin { ExternalAccessible := 'False'; ExternalVisible := 'False'; ExternalWritable := 'False'} : Int;
      si_RequestedPosition { ExternalAccessible := 'False'; ExternalVisible := 'False'; ExternalWritable := 'False'} : Int;
      si_LoopCounterPositions { ExternalAccessible := 'False'; ExternalVisible := 'False'; ExternalWritable := 'False'} : Int;   // Loopcounter positions
      si_LoopCounterDestinations { ExternalAccessible := 'False'; ExternalVisible := 'False'; ExternalWritable := 'False'} : Int;   // Loopcounter destinations
      si_NumberOfPositons { ExternalAccessible := 'False'; ExternalVisible := 'False'; ExternalWritable := 'False'} : Int;   // Number of positions in the search area
      si_NumberOfDestinations { ExternalAccessible := 'False'; ExternalVisible := 'False'; ExternalWritable := 'False'} : Int;   // Number of destinations per position
      sx_NewGinFound { ExternalAccessible := 'False'; ExternalVisible := 'False'; ExternalWritable := 'False'} : Bool;   // Memory to start searching
   END_VAR


BEGIN
	(*
	----------------------------------------------------------------------------------------

	Version history:
	Date        | Version   | Author        | Remark
	----------------------------------------------------------------------------------------
	10-09-2019  | 2.0       | F.Baten       | Doubled search loop and added comment
	12/11/2019  | 3.0       | P.Majka       | 3.0 MHS library release TIA 15.1
	08/01/2020  | 3.1       | F.Baten       | When no destination is given, also go to default direction
	15/01/2019  | 3.2       | L.Klar        | GIN record structure updated, parcel destination remapped
	19/10/2020  | 3.3       | L.Klar        | Double search loop reprogrammed, issue with default position
	07/12/2020  | 3.4       | L.Klar        | GIN greater than zero condition added to region 2
	21/02/2023  | 4.0       | F.Baten       | 4.0 Release TIA 17.5
	*)


	REGION 1 - Determine size OF search area

	    #si_NumberOfPositons := "FC_GetNrOfArrayEl"(#iqa_DBDestination);
	    #si_NumberOfDestinations := "FC_GetNrOfArrayEl"(#iqa_DBDestination[1].Destination);

	END_REGION

	REGION 2 - Get GIN from tracking DB
	    // There is a value in the tracking data on the decision point which is not '0' or equal to the previous GIN

	    IF (#iqa_TrackingData[#iqUDT_VSUInterface.Decisionpoint] <> 0) AND (#iqa_TrackingData[#iqUDT_VSUInterface.Decisionpoint] <> #si_PreviousGin)
	    THEN
	        #si_Gin := #iqa_TrackingData[#iqUDT_VSUInterface.Decisionpoint];
	        #sx_NewGinFound := TRUE;
	    END_IF;

	END_REGION

	REGION 2 - Get destination from GIN DB
	    // If new GIN has been detected, get destination from its GIN record

	    IF #sx_NewGinFound AND #si_Gin > 0
	    THEN
	        #sdi_RequestedDestination := "DB_GIN".GIN[#si_Gin].General.Destination[0];
	        #si_PreviousGin := #si_Gin;
	        #si_Gin := 0;
	        #iqUDT_VSUInterface.RequestedPosition := 0;
	    END_IF;

	END_REGION

	REGION 3 - Get requested position when new GIN is found
	    IF #sx_NewGinFound
	    THEN
	        // If destination is different than 0, find a position in destination arrays. Otherwise, requested position is set to default.
	        IF #sdi_RequestedDestination <> 0 THEN
	            FOR #si_LoopCounterPositions := 1 TO #si_NumberOfPositons BY 1 DO
	                FOR #si_LoopCounterDestinations := 0 TO (#si_NumberOfDestinations - 1) BY 1 DO
	                    IF #iqa_DBDestination[#si_LoopCounterPositions].Destination[#si_LoopCounterDestinations] = #sdi_RequestedDestination
	                    THEN
	                        #si_RequestedPosition := #si_LoopCounterPositions;
	                        EXIT;
	                    END_IF;
	                END_FOR;
	                // Position found
	                IF #si_RequestedPosition <> 0
	                THEN
	                    #iqUDT_VSUInterface.RequestedPosition := #si_RequestedPosition;
	                    #sx_NewGinFound := FALSE;
	                    #si_RequestedPosition := 0;
	                    EXIT;
	                END_IF;
	            END_FOR;
	        ELSE
	            // Default position
	            #sx_NewGinFound := FALSE;
	            #iqUDT_VSUInterface.RequestedPosition := 99;
	            #si_RequestedPosition := 0;
	        END_IF;
	    END_IF;
	END_REGION
END_FUNCTION_BLOCK

FUNCTION_BLOCK "FB_InchingBulk"
{ S7_Optimized_Access := 'TRUE' }
VERSION : 0.1
// ATTRIBUTES
// AUTO_NUMBER = True
// BLOCK_NUMBER = 13
// END_ATTRIBUTES
   VAR_INPUT
      ix_PECUp { ExternalAccessible := 'False'; ExternalVisible := 'False'; ExternalWritable := 'False'} : Bool;   // PEC Sum signal from upstream conveyor
      ix_InchingActive { ExternalAccessible := 'False'; ExternalVisible := 'False'; ExternalWritable := 'False'} : Bool;   // If TRUE inching is activate
      ix_ClearCommand { ExternalAccessible := 'False'; ExternalVisible := 'False'; ExternalWritable := 'False'} : Bool;   // Command to clear full status
      ix_DownstreamFull { ExternalAccessible := 'False'; ExternalVisible := 'False'; ExternalWritable := 'False'} : Bool;   // TRUE if downstream conveyors are full
      ii_OnDelayGap { ExternalAccessible := 'False'; ExternalVisible := 'False'; ExternalWritable := 'False'} : DInt;   // Distance to conveyor release [mm]
      ii_InchingGap { ExternalAccessible := 'False'; ExternalVisible := 'False'; ExternalWritable := 'False'} : DInt;   // Inching distance [mm]
      ii_Displacement_Upstream { ExternalAccessible := 'False'; ExternalVisible := 'False'; ExternalWritable := 'False'} : Int;   // Upstream conveyor displacement
      ii_Displacement { ExternalAccessible := 'False'; ExternalVisible := 'False'; ExternalWritable := 'False'} : Int;   // Inching conveyor displacement
   END_VAR

   VAR_OUTPUT
      qx_ExternalRequestHold { ExternalAccessible := 'False'; ExternalVisible := 'False'; ExternalWritable := 'False'} : Bool;   // External output to request conveyor hold
      qx_Full { ExternalAccessible := 'False'; ExternalVisible := 'False'; ExternalWritable := 'False'} : Bool;   // Inching conveyor is full status
   END_VAR

   VAR
      sUDT_Status { ExternalAccessible := 'False'; ExternalVisible := 'False'; ExternalWritable := 'False'; S7_SetPoint := 'False'} : "UDT_InchingStatus";
      sUDT_StatusOld { ExternalAccessible := 'False'; ExternalVisible := 'False'; ExternalWritable := 'False'; S7_SetPoint := 'False'} : "UDT_InchingStatus";
      F_TRIG_PECEoSUp {InstructionName := 'F_TRIG'; LibVersion := '1.0'; ExternalAccessible := 'False'; ExternalVisible := 'False'; ExternalWritable := 'False'; S7_SetPoint := 'False'} : F_TRIG;   // Falling edge trigger PEC EoS
      si_ActualInchingGap { ExternalAccessible := 'False'; ExternalVisible := 'False'; ExternalWritable := 'False'} : Int;   // Distance to request hold
      si_ActualOnGap { ExternalAccessible := 'False'; ExternalVisible := 'False'; ExternalWritable := 'False'} : Int;   // Distance to conveyor release
      sx_StartRelease { ExternalAccessible := 'False'; ExternalVisible := 'False'; ExternalWritable := 'False'} : Bool;   // Conveyor release
      sx_ConveyorFull { ExternalAccessible := 'False'; ExternalVisible := 'False'; ExternalWritable := 'False'} : Bool;
   END_VAR


BEGIN
	(*
	----------------------------------------------------------------------------------------

	Version history:
	Date        | Version   | Author        | Remark
	----------------------------------------------------------------------------------------
	01/04/2021  | 1.0       | M.Kocot       | first release TIA 16
	08/04/2021  | 1.1       | H.Rutkwoski   | Added status full
	14/08/2021  | 1.2       | M. Jager      | Reset sx_full when inching is not active
	21/02/2023  | 4.0       | F.Baten       | 4.0 Release TIA 17.5
	12/03/2024  | 4.1       | S. Nieswiec   | Removed underscore from function name
	*)

	REGION 1 - Triggers

	    // Falling edge trigger PEC EoS.
	    #F_TRIG_PECEoSUp(CLK := #ix_PECUp);

	END_REGION


	REGION 2 - Inching
	    // Statement section REGION

	    #qx_ExternalRequestHold := #ix_InchingActive;

	    IF #F_TRIG_PECEoSUp.Q AND #ix_InchingActive THEN
	        #si_ActualOnGap := DINT_TO_INT(#ii_OnDelayGap / 10);
	        #si_ActualInchingGap := DINT_TO_INT(#ii_InchingGap / 10);

	    END_IF;

	    IF #si_ActualOnGap > 0 THEN

	        #si_ActualOnGap := #si_ActualOnGap - #ii_Displacement_Upstream;

	    END_IF;

	    IF #ix_PECUp AND #si_ActualInchingGap > 0 THEN
	        #si_ActualInchingGap := #si_ActualInchingGap - #ii_Displacement;
	    END_IF;

	    IF #si_ActualOnGap <= 0
	        OR #sx_StartRelease
	    THEN
	        #sx_StartRelease := TRUE;
	    END_IF;

	    IF #si_ActualInchingGap <= 0
	    THEN
	        #sx_StartRelease := FALSE;
	    END_IF;

	    IF #sx_StartRelease THEN
	        #qx_ExternalRequestHold := FALSE;
	    END_IF;

	END_REGION

	REGION 3 - Internal status - convayor full

	    // Set conveyor status to full when:
	    IF #ix_InchingActive                     // inching is active
	        AND #ix_DownstreamFull               // downstream is full
	        AND NOT #ix_ClearCommand             // there is no clear command active
	    THEN
	        #sx_ConveyorFull := TRUE;
	    END_IF;

	    // Set conveyor status to NOT full when:
	    IF (#ix_InchingActive                   // Inching is active
	        AND #ix_ClearCommand                // clear command is active
	        AND NOT #ix_DownstreamFull)         // downstream is NOT full)
	        OR NOT #ix_InchingActive            // OR Inching isnt active
	    THEN
	        #sx_ConveyorFull := FALSE;
	    END_IF;

	END_REGION


	REGION 4 - Status

	    // Convsyor is full status
	    #sUDT_Status.Full := #sx_ConveyorFull;

	    #sUDT_Status.Active := #ix_InchingActive;

	    // Status update on change.
	    IF #sUDT_StatusOld <> #sUDT_Status
	    THEN
	        #qx_Full := #sUDT_Status.Full;
	        #sUDT_StatusOld := #sUDT_Status;
	    END_IF;

	END_REGION


END_FUNCTION_BLOCK

FUNCTION_BLOCK "FB_MainControlPanel"
TITLE = Main Control Panel Cabinet Block
{ S7_Optimized_Access := 'TRUE' }
AUTHOR : CesarLeite
VERSION : 3.0
// ATTRIBUTES
// AUTO_NUMBER = True
// BLOCK_NUMBER = 253
// END_ATTRIBUTES
   VAR_INPUT
      is_PNPNCouplerDeviceName { ExternalAccessible := 'False'; ExternalVisible := 'False'; ExternalWritable := 'False'} : String;   //  Name of the PN PN coupler device
      is_SingulatorCouplerDeviceName { ExternalAccessible := 'False'; ExternalVisible := 'False'; ExternalWritable := 'False'} : String;   //  Name of the Singulator coupler device
      is_IOModulePNDeviceName { ExternalAccessible := 'False'; ExternalVisible := 'False'; ExternalWritable := 'False'} : String := '';   //  Name of the ET200sp device
      is_ScalanceSwitchName { ExternalAccessible := 'False'; ExternalVisible := 'False'; ExternalWritable := 'False'} : String;   // Name of the Scalance Switch
      ii_Racksize { ExternalAccessible := 'False'; ExternalVisible := 'False'; ExternalWritable := 'False'} : Int;   //  Number off slots present in the rack
      ix_UPSOk { ExternalAccessible := 'False'; ExternalVisible := 'False'; ExternalWritable := 'False'} : Bool;   //  TRUE if Unit Power Supply with no faults
      ix_NoFireAlarmActive { ExternalAccessible := 'False'; ExternalVisible := 'False'; ExternalWritable := 'False'} : Bool;   //  TRUE if Fire alarm is not active
      ix_24V201T1 { ExternalAccessible := 'False'; ExternalVisible := 'False'; ExternalWritable := 'False'} : Bool;   //  TRUE if power supply has no warning
      ix_CBTripped101F4 { ExternalAccessible := 'False'; ExternalVisible := 'False'; ExternalWritable := 'False'} : Bool;   //  TRUE if MCP circuit breaker is tripped
      ix_CBTripped102F1 { ExternalAccessible := 'False'; ExternalVisible := 'False'; ExternalWritable := 'False'} : Bool;   //  TRUE if MCP circuit breaker is not tripped
      ix_CBTripped201F1 { ExternalAccessible := 'False'; ExternalVisible := 'False'; ExternalWritable := 'False'} : Bool;   //  TRUE if MCP circuit breaker is not tripped
      ix_CBTripped205F5 { ExternalAccessible := 'False'; ExternalVisible := 'False'; ExternalWritable := 'False'} : Bool;   //  TRUE if MCP circuit breaker is not tripped
      ix_ScalanceSwitchStatus { ExternalAccessible := 'False'; ExternalVisible := 'False'; ExternalWritable := 'False'} : Bool;   // TRUE if the scalance switch is Healthy
      ix_SimulationModeActive { ExternalAccessible := 'False'; ExternalVisible := 'False'; ExternalWritable := 'False'} : Bool;   //  TRUE if simulation is active
      ix_SingulatorCouplerAvailable { ExternalAccessible := 'False'; ExternalVisible := 'False'; ExternalWritable := 'False'} : Bool;   //  TRUE if singulator coulper available in cabinet
      ix_ExternalScan { ExternalAccessible := 'False'; ExternalVisible := 'False'; ExternalWritable := 'False'} : Bool;   //  External scan
      ix_HardwareOk { ExternalAccessible := 'False'; ExternalVisible := 'False'; ExternalWritable := 'False'} : Bool;   //  TRUE when  hardware is Ok
   END_VAR

   VAR_OUTPUT
      qUDT_HMIStatus { ExternalAccessible := 'False'; ExternalVisible := 'False'; ExternalWritable := 'False'} : "UDT_MainControlPanelStatus";   //  HMI status structure
      qUDT_Status { ExternalAccessible := 'False'; ExternalVisible := 'False'; ExternalWritable := 'False'} : "UDT_CommonStatus";   //  Common status structure
   END_VAR

   VAR_IN_OUT
      iqUDT_Statistics : "UDT_MainControlPanelStatistics";   //  Statistics structure
      iqUDT_EquipmentControl : "UDT_EquipmentControl";   //  Equipment control structure
   END_VAR

   VAR
      sUDT_PNCouplerPNDevice { ExternalAccessible := 'False'; ExternalVisible := 'False'; ExternalWritable := 'False'; S7_SetPoint := 'False'} : "UDT_PNDevice";   //  PN device structure
      sUDT_ScalanceSwitchDevice { ExternalAccessible := 'False'; ExternalVisible := 'False'; ExternalWritable := 'False'; S7_SetPoint := 'False'} : "UDT_PNDevice";   // Scalance Switch device structure
      sUDT_SingulatorCouplerPNDevice { ExternalAccessible := 'False'; ExternalVisible := 'False'; ExternalWritable := 'False'; S7_SetPoint := 'False'} : "UDT_PNDevice";   //  PN device structure
      sUDT_CommonStatus { ExternalAccessible := 'False'; ExternalVisible := 'False'; ExternalWritable := 'False'; S7_SetPoint := 'False'} : "UDT_CommonStatus";   //  Common status structure
      sUDT_CommonStatusOld { ExternalAccessible := 'False'; ExternalVisible := 'False'; ExternalWritable := 'False'; S7_SetPoint := 'False'} : "UDT_CommonStatus";   //  Auxiliary status structure
      sUDT_MasterControlPanelRIOStatus { ExternalAccessible := 'False'; ExternalVisible := 'False'; ExternalWritable := 'False'; S7_SetPoint := 'False'} : "UDT_CommonStatus";   //  Common status structure
      sUDT_HMIStatus { ExternalAccessible := 'False'; ExternalVisible := 'False'; ExternalWritable := 'False'; S7_SetPoint := 'False'} : "UDT_MainControlPanelStatus";   //  MCP status UDT
      sUDT_RIOStatistics { ExternalAccessible := 'False'; ExternalVisible := 'False'; ExternalWritable := 'False'; S7_SetPoint := 'False'} : "UDT_RIOStatistics";   //  Statistics structure
      sUDT_MasterControlPanelRIOHMIStatus { ExternalAccessible := 'False'; ExternalVisible := 'False'; ExternalWritable := 'False'; S7_SetPoint := 'False'} : "UDT_RIOStatus";   // MCP I/O Module status
      sFB_MasterControlPanelRIO { ExternalAccessible := 'False'; ExternalVisible := 'False'; ExternalWritable := 'False'; S7_SetPoint := 'False'} : "FB_RIO";   // MCP I/O module fucntion block
      sFB_TimerOnOffDelayCheckSupply { ExternalAccessible := 'False'; ExternalVisible := 'False'; ExternalWritable := 'False'; S7_SetPoint := 'False'} : "FB_TimerOnOffDelay";   //  MHS "TimerOnOffDelay" - to delay time for VFD supply contactor
      sa_PNCouplerPortsStatus { ExternalAccessible := 'False'; ExternalVisible := 'False'; ExternalWritable := 'False'} : Array[1..8] of Bool;   // TRUE when specific PN coupler port has an error
      sa_SingulatorPortsStatus { ExternalAccessible := 'False'; ExternalVisible := 'False'; ExternalWritable := 'False'} : Array[1..8] of Bool;   // TRUE when specific IO module port has an error
      sa_ScalanceSwitchStatus { ExternalAccessible := 'False'; ExternalVisible := 'False'; ExternalWritable := 'False'} : Array[1..8] of Bool;   // TRUE when specific IO module port has an error
      sa_Status { ExternalAccessible := 'False'; ExternalVisible := 'False'; ExternalWritable := 'False'} : Struct   //  Status structure
         ErrorCode { ExternalAccessible := 'False'; ExternalVisible := 'False'; ExternalWritable := 'False'} : Struct   //  Error code structure
            ModuleState { ExternalAccessible := 'False'; ExternalVisible := 'False'; ExternalWritable := 'False'} : Int;   //  Siemens "ModuleState" error code
         END_STRUCT;
      END_STRUCT;
      sR_Trig_UPS {InstructionName := 'R_TRIG'; LibVersion := '1.0'; ExternalAccessible := 'False'; ExternalVisible := 'False'; ExternalWritable := 'False'; S7_SetPoint := 'False'} : R_TRIG;   //  Rise trigger when a UPS fault occurs
      sR_Trig_PNCoupler {InstructionName := 'R_TRIG'; LibVersion := '1.0'; ExternalAccessible := 'False'; ExternalVisible := 'False'; ExternalWritable := 'False'; S7_SetPoint := 'False'} : R_TRIG;   //  Rise trigger when a PN/PN Coupler fault occurs
      sR_Trig_ProSoftCoupler {InstructionName := 'R_TRIG'; LibVersion := '1.0'; ExternalAccessible := 'False'; ExternalVisible := 'False'; ExternalWritable := 'False'; S7_SetPoint := 'False'} : R_TRIG;   //  Rise trigger when a ProSoft Coupler fault occurs
      sR_Trig_MainRackModule {InstructionName := 'R_TRIG'; LibVersion := '1.0'; ExternalAccessible := 'False'; ExternalVisible := 'False'; ExternalWritable := 'False'; S7_SetPoint := 'False'} : R_TRIG;   //  Rise trigger when there is an error on the mainrack modules
      sR_Trig_FireAlarm {InstructionName := 'R_TRIG'; LibVersion := '1.0'; ExternalAccessible := 'False'; ExternalVisible := 'False'; ExternalWritable := 'False'; S7_SetPoint := 'False'} : R_TRIG;   //  Rise trigger when a Fire alarm fault occurs
      sR_Trig_ScalanceSwitchStatus {InstructionName := 'R_TRIG'; LibVersion := '1.0'; ExternalAccessible := 'False'; ExternalVisible := 'False'; ExternalWritable := 'False'; S7_SetPoint := 'False'} : R_TRIG;   //  Rise trigger when a scalance switch status is not healthy
      sR_Trig_ScalanceSwitch {InstructionName := 'R_TRIG'; LibVersion := '1.0'; ExternalAccessible := 'False'; ExternalVisible := 'False'; ExternalWritable := 'False'; S7_SetPoint := 'False'} : R_TRIG;   //  Rise trigger when a scalance switch fault occurs
      sR_Trig_24V_201T1 {InstructionName := 'R_TRIG'; LibVersion := '1.0'; ExternalAccessible := 'False'; ExternalVisible := 'False'; ExternalWritable := 'False'; S7_SetPoint := 'False'} : R_TRIG;   //  Rise trigger when a 201T1 circuit braker tripped
      sR_Trig_CB_Tripped_101F4 {InstructionName := 'R_TRIG'; LibVersion := '1.0'; ExternalAccessible := 'False'; ExternalVisible := 'False'; ExternalWritable := 'False'; S7_SetPoint := 'False'} : R_TRIG;   //  Rise trigger when a 101F4 circuit braker tripped
      sR_Trig_CB_Tripped_102F1 {InstructionName := 'R_TRIG'; LibVersion := '1.0'; ExternalAccessible := 'False'; ExternalVisible := 'False'; ExternalWritable := 'False'; S7_SetPoint := 'False'} : R_TRIG;   //  Rise trigger when a 102F1 circuit braker tripped
      sR_Trig_CB_Tripped_201F1 {InstructionName := 'R_TRIG'; LibVersion := '1.0'; ExternalAccessible := 'False'; ExternalVisible := 'False'; ExternalWritable := 'False'; S7_SetPoint := 'False'} : R_TRIG;   //  Rise trigger when a 201F1 circuit braker tripped
      sR_Trig_CB_Tripped_205F5 {InstructionName := 'R_TRIG'; LibVersion := '1.0'; ExternalAccessible := 'False'; ExternalVisible := 'False'; ExternalWritable := 'False'; S7_SetPoint := 'False'} : R_TRIG;   //  Rise trigger when a 205F5 circuit braker tripped
      sx_RackCheck { ExternalAccessible := 'False'; ExternalVisible := 'False'; ExternalWritable := 'False'} : Bool;   //  Start checking the mainrack
      sx_PowerOk { ExternalAccessible := 'False'; ExternalVisible := 'False'; ExternalWritable := 'False'} : Bool;   //  True = External Power OK
   END_VAR

   VAR_TEMP
      ts_Configured : Array[0..127] of Bool;   //  Configured structure
      ts_Exist : Array[0..127] of Bool;   //  Exits structure
      ts_Error : Array[0..127] of Bool;   //  Error structure
      ti_Racksize : Int;   //  The limited size of the rack
      ti_ModuleNr : Int;   //  The number of the module being processed
   END_VAR

   VAR CONSTANT
      ci_PowerSupplyDelayTime : UInt := 4000;   //  Power supply delay time
      cui_LADDR : UInt := 32;   //  Local~Device
      cui_ConfiguredDevicesMode : UInt := 1;   //  Scan mode of configured devices
      cui_ExistingDevicesMode : UInt := 4;   //  Scan mode of existing devices
      cui_DevicesErrorMode : UInt := 2;   //  Scan mode of devices error
      ci_NumberOfProfinetPorts : Int := 2;   // Number of Profinet ports in device
      ci_RackMaximumSize : Int := 31;
      ci_RackMinimumSize : Int := 4;
   END_VAR


BEGIN
	(*
	----------------------------------------------------------------------------------------

	Version history:
	Date        | Version   | Author        | Remark
	----------------------------------------------------------------------------------------
	17/09/2019  | 2.0       | C.Leite       | first release TIA 15.1
	14/10/2019  | 2.1       | L.Klar        | Updated status structure
	16/10/2019  | 2.2       | S. Deulkar    | USed FC_GetDevice PN to create PN error
	30/10/2019  | 2.3       | M. Kurpiers   | Regions renumbering
	12/11/2019  | 3.0       | P.Majka       | 3.0 MHS library release TIA 15.1
	04/11/2019  | 3.1       | F.Baten       | Region 4: ix_SimulationModeActive rearranged to correct position
	25/02/2020  | 3.2       | S. Deulkar    | Modified to update ststus output every cycle
	06/05/2020  | 3.3       | F.Baten       | New UDT_MCPStatus
	24/06/2020  | 3.4       | F.Baten       | Mainrack module state function added
	29/06/2020  | 3.5       | F.Baten       | Changed statistics for Mainrack modules
	07/07/2020  | 3.6       | S.Theocharis  | Change HMI status to IO
	09/07/2020  | 3.7       | S.Theocharis  | Bug fix in status update. Initialize static status instead output status
	20/07/2020  | 3.8       | K.Pokorski    | Bug fix in PLC module status update. Change HMI status from InOut to Out
	03/11/2020  | 3.9       | K.Pokorski    | Profinet ports diagnostics added
	14/04/2021  | 3.10      | H.Rutkowski   | FB_RIO for MCP Remote IO integarted into the function
	                                        | Added new inputs from MCP Remote IO with the corresponding errors, statuses and statistics
	16/07/2021  | 3.11      | M. roijen     | Bug fix reset errors PN-PN_PNSlaveWarning and PS_201T4_Warning
	14-08-2021  | 3.12      | S. Deulkar    | added set profinet scan when PLC has error region 5
	16/02/2022  | 3.13      | M.Piela       | FedEx release
	11/05/2022  | 3.14      | M.Singh       | Changes equivalant to name change in UDT MCP status
	21/02/2023  | 4.0       | F.Baten       | 4.0 Release TIA 17.5
	*)


	REGION 1 – Get Device Profinet information

	    // PN Coupler
	    "FC_GetDevicePN"(is_PNDeviceName := #is_PNPNCouplerDeviceName,
	                     ix_SimulationModeActive := #ix_SimulationModeActive,
	                     iqUDT_PND := #sUDT_PNCouplerPNDevice);


	    "FC_GetPNPortStatus"(ii_NumberOfPorts := #ci_NumberOfProfinetPorts,
	                         iUDT_DevicePNInfo := #sUDT_PNCouplerPNDevice,
	                         qa_PortFault => #sa_PNCouplerPortsStatus);

	    // Singulator PN coupler

	    "FC_GetDevicePN"(is_PNDeviceName := #is_SingulatorCouplerDeviceName,
	                     ix_SimulationModeActive := #ix_SimulationModeActive,
	                     iqUDT_PND := #sUDT_SingulatorCouplerPNDevice);

	    "FC_GetPNPortStatus"(ii_NumberOfPorts := #ci_NumberOfProfinetPorts,
	                         iUDT_DevicePNInfo := #sUDT_SingulatorCouplerPNDevice,
	                         qa_PortFault => #sa_SingulatorPortsStatus);

	    // IO Module - Region 4

	    //Scalance switch

	    "FC_GetDevicePN"(is_PNDeviceName := #is_ScalanceSwitchName,
	                     ix_SimulationModeActive := #ix_SimulationModeActive,
	                     iqUDT_PND := #sUDT_ScalanceSwitchDevice);

	    "FC_GetPNPortStatus"(ii_NumberOfPorts := #ci_NumberOfProfinetPorts,
	                         iUDT_DevicePNInfo := #sUDT_ScalanceSwitchDevice,
	                         qa_PortFault => #sa_ScalanceSwitchStatus);

	END_REGION

	REGION 2 – Triggers

	    // Rise trigger UPS status
	    #sR_Trig_UPS(CLK := #sUDT_HMIStatus.Specific.UPSSwitchTripped);

	    // Rise trigger Fire alarm status
	    #sR_Trig_FireAlarm(CLK := #sUDT_HMIStatus.Specific.FireAlarmActive);

	    #sR_Trig_24V_201T1(CLK := #sUDT_HMIStatus.Specific.PS_201T1_Tripped);

	    #sR_Trig_CB_Tripped_101F4(CLK := #sUDT_HMIStatus.Specific."230VAC_CB101F4Tripped");

	    #sR_Trig_CB_Tripped_102F1(CLK := #sUDT_HMIStatus.Specific."230VAC_CB102F1Tripped");

	    #sR_Trig_CB_Tripped_201F1(CLK := #sUDT_HMIStatus.Specific."24VDC_CB201F1Tripped");

	    #sR_Trig_CB_Tripped_205F5(CLK := #sUDT_HMIStatus.Specific."24VDC_CB205F5Tripped");

	    #sR_Trig_ScalanceSwitchStatus(CLK := #sUDT_HMIStatus.Specific.ScalanceSwitchStatus);

	    // Rise trigger PN/PN coupler status
	    #sR_Trig_PNCoupler(CLK := #sUDT_HMIStatus.Specific."PN_PN_MSP_PNSlaveNotOnline" OR #sUDT_HMIStatus.Specific."PN_PN_MSP_PNSlaveError");

	    // Rise trigger Singulator coupler status
	    #sR_Trig_ProSoftCoupler(CLK := #sUDT_HMIStatus.Specific.Singulator_PNSlaveNotOnline OR #sUDT_HMIStatus.Specific.Singulator_PNSlaveError);

	    // Rise trigger Scalance switch status
	    #sR_Trig_ScalanceSwitch(CLK := #sUDT_HMIStatus.Specific.ScalanceSwitchPNSlaveNotOnline OR #sUDT_HMIStatus.Specific.ScalanceSwitchPNSlaveError);

	    // rising trigger main rack module status
	    #sR_Trig_MainRackModule(CLK := #sUDT_HMIStatus.Specific.RackSlotError[0]);

	END_REGION

	REGION 3 – Reset error
	    // All faults are reset when the reset input is true

	    IF #iqUDT_EquipmentControl.Command.Reset
	    THEN
	        #sUDT_HMIStatus.Specific.ScalanceSwitchStatus := FALSE;
	        #sUDT_HMIStatus.Specific.PS_201T1_Tripped := FALSE;
	        #sUDT_HMIStatus.Specific."230VAC_CB101F4Tripped" := FALSE;
	        #sUDT_HMIStatus.Specific."230VAC_CB102F1Tripped" := FALSE;
	        #sUDT_HMIStatus.Specific."24VDC_CB201F1Tripped" := FALSE;
	        #sUDT_HMIStatus.Specific."24VDC_CB205F5Tripped" := FALSE;
	        #sUDT_HMIStatus.Specific.FireAlarmActive := FALSE;
	        #sUDT_HMIStatus.Specific.UPSSwitchTripped := FALSE;
	        #sUDT_HMIStatus.Specific."PN_PN_MSP_PNSlaveNotOnline" := FALSE;
	        #sUDT_HMIStatus.Specific."PN_PN_MSP_PNSlaveError" := FALSE;
	        #sUDT_HMIStatus.Specific."PN_PN_MSP_PNSlaveWarning" := FALSE;
	        #sUDT_HMIStatus.Specific.ScalanceSwitchPNSlaveError := FALSE;
	        #sUDT_HMIStatus.Specific.ScalanceSwitchPNSlaveNotOnline := FALSE;
	        #sUDT_HMIStatus.Specific.ScalanceSwitchPNSlaveWarning := FALSE;
	        #sUDT_HMIStatus.Specific.Singulator_PNSlaveNotOnline := FALSE;
	        #sUDT_HMIStatus.Specific.Singulator_PNSlaveError := FALSE;
	        #sUDT_HMIStatus.Specific.Singulator_PNSlaveWarning := FALSE;

	    END_IF;

	END_REGION

	REGION 4 – Master control panel remote input output

	    #sFB_MasterControlPanelRIO(ix_24VOk := TRUE,
	                               ix_SimulationModeActive := #ix_SimulationModeActive,
	                               is_ET200spPNDeviceName := #is_IOModulePNDeviceName,
	                               qUDT_HMIStatus => #sUDT_MasterControlPanelRIOHMIStatus,
	                               qUDT_Status => #sUDT_MasterControlPanelRIOStatus,
	                               iqUDT_EquipmentControl := #iqUDT_EquipmentControl,
	                               iqUDT_Statistics := #sUDT_RIOStatistics);

	    #sUDT_HMIStatus.Specific.IOModuleSlotError := #sUDT_MasterControlPanelRIOHMIStatus.Specific.ET200sp_ErrorModule;

	    #sUDT_HMIStatus.Specific.IOModule_PNSlaveError := #sUDT_MasterControlPanelRIOHMIStatus.Specific.PNSlaveError;

	    #sUDT_HMIStatus.Specific.IOModule_PNSlaveNotOnline := false;// #s_UDT_MCP_RIO_HMIStatus.Specific.PNSlaveNotOnline;

	    #sUDT_HMIStatus.Specific.IOModule_PNSlaveWarning := #sUDT_MasterControlPanelRIOHMIStatus.Specific.PNSlaveWarning;

	    #iqUDT_Statistics.IOModuleCouplerFault := #sUDT_RIOStatistics.PNSlaveError;

	END_REGION

	REGION 5 – Scan request
	    // Start scan when request from diagnostic OB, First PLC cycle or External scan request
	    IF ("DB_Memory".ScanMainRack
	        OR "DB_Memory".FirstScan
	        OR #ix_ExternalScan)
	    THEN
	        #sx_RackCheck := TRUE;
	        "DB_Memory".ScanMainRack := FALSE;
	    END_IF;

	    //Set the profinet scan when the error on the PLC occour
	    IF #sR_Trig_MainRackModule.Q
	    THEN
	        "DB_Memory".ScanProfinet := TRUE;
	    END_IF;

	END_REGION

	REGION 6 – Modules states update

	    // When in the fault/diagnostic OB 82,83,86 the bit is set, the function activates
	    IF #sx_RackCheck
	    THEN

	        REGION 6.1 - Check racksize
	            // limiting the racksize between 4 and 31 positions
	            #ti_Racksize := #ii_Racksize;
	            IF #ti_Racksize > #ci_RackMaximumSize
	            THEN
	                #ti_Racksize := #ci_RackMaximumSize;
	            END_IF;
	            IF #ti_Racksize < #ci_RackMinimumSize
	            THEN
	                #ti_Racksize := #ci_RackMinimumSize;
	            END_IF;
	        END_REGION

	        REGION 6.2 - Get the module from the io system

	            // Get the module state from the mainrack
	            #sa_Status.ErrorCode.ModuleState := ModuleStates(LADDR := #cui_LADDR,
	                                                             MODE := #cui_ConfiguredDevicesMode,
	                                                             STATE := #ts_Configured);

	            #sa_Status.ErrorCode.ModuleState := ModuleStates(LADDR := #cui_LADDR,
	                                                             MODE := #cui_ExistingDevicesMode,
	                                                             STATE := #ts_Exist);

	            #sa_Status.ErrorCode.ModuleState := ModuleStates(LADDR := #cui_LADDR,
	                                                             MODE := #cui_DevicesErrorMode,
	                                                             STATE := #ts_Error);
	        END_REGION

	        REGION 6.3 - Set the error
	            // A loop operating on all modules if configured for the selected racksize
	            // If a device is configured and not existing or in error, the error bit is set
	            FOR #ti_ModuleNr := 0 TO #ti_Racksize
	            DO
	                IF (#ts_Configured[#ti_ModuleNr])
	                    AND ((NOT #ts_Exist[#ti_ModuleNr])
	                    OR (#ts_Error[#ti_ModuleNr]))
	                THEN
	                    #sUDT_HMIStatus.Specific.RackSlotError[#ti_ModuleNr] := TRUE;
	                ELSE
	                    IF #iqUDT_EquipmentControl.Command.Reset
	                    THEN
	                        #sUDT_HMIStatus.Specific.RackSlotError[#ti_ModuleNr] := FALSE;
	                    END_IF;
	                END_IF;
	            END_FOR;
	        END_REGION

	    END_IF;

	END_REGION

	REGION 7 - Reset the Rackcheck

	    // If the main module is not signalling an error the rackcheck is reset
	    IF #sx_RackCheck AND NOT #sUDT_HMIStatus.Specific.RackSlotError[0]
	    THEN
	        #sx_RackCheck := False;
	    END_IF;
	END_REGION

	REGION 8 - Faults monitoring

	    // Hardware will only be available after the delay, so the device has time for the initialization
	    #sFB_TimerOnOffDelayCheckSupply(iudi_OnDelayTime := #ci_PowerSupplyDelayTime,
	                                    ix_SignalToDelay := #ix_CBTripped205F5,//   //#ix_24VDCOk,
	                                    qx_DelayedSignal => #sx_PowerOk);

	    // check if PN PN coupler is online
	    IF (NOT "DB_ProfinetDiagnostic".ProfinetNetworks[#sUDT_PNCouplerPNDevice.PNNetworknumber].DeviceStatus[#sUDT_PNCouplerPNDevice.PNDeviceNumber].DeviceState.Exist
	        OR NOT #sUDT_PNCouplerPNDevice.PNDeviceFound)
	        AND #sx_PowerOk
	        AND NOT #ix_SimulationModeActive
	    THEN
	        #sUDT_HMIStatus.Specific."PN_PN_MSP_PNSlaveNotOnline" := TRUE;
	    END_IF;

	    // Check if PN ports are healthy
	    IF #sa_PNCouplerPortsStatus[1] XOR #sa_PNCouplerPortsStatus[2] THEN
	        #sUDT_HMIStatus.Specific."PN_PN_MSP_PNSlaveWarning" := TRUE;
	    END_IF;


	    // check if PN PN coupler has an error
	    IF "DB_ProfinetDiagnostic".ProfinetNetworks[#sUDT_PNCouplerPNDevice.PNNetworknumber].DeviceStatus[#sUDT_PNCouplerPNDevice.PNDeviceNumber].DeviceState.Error
	        AND #sx_PowerOk
	        AND NOT #ix_SimulationModeActive
	        AND NOT #sUDT_HMIStatus.Specific."PN_PN_MSP_PNSlaveWarning"
	    THEN
	        #sUDT_HMIStatus.Specific."PN_PN_MSP_PNSlaveError" := TRUE;
	    END_IF;

	    // check if Scalance Switch is online
	    IF (NOT "DB_ProfinetDiagnostic".ProfinetNetworks[#sUDT_ScalanceSwitchDevice.PNNetworknumber].DeviceStatus[#sUDT_ScalanceSwitchDevice.PNDeviceNumber].DeviceState.Exist
	        OR NOT #sUDT_ScalanceSwitchDevice.PNDeviceFound)
	        AND #sx_PowerOk
	        AND NOT #ix_SimulationModeActive
	    THEN
	        #sUDT_HMIStatus.Specific.ScalanceSwitchPNSlaveNotOnline := TRUE;
	    END_IF;

	    // Check if Scalance Switch ports are healthy
	    IF #sa_ScalanceSwitchStatus[1] XOR #sa_ScalanceSwitchStatus[2] THEN
	        #sUDT_HMIStatus.Specific."PN_PN_MSP_PNSlaveWarning" := TRUE;
	    END_IF;


	    // check if Scalance Switch has an error
	    IF "DB_ProfinetDiagnostic".ProfinetNetworks[#sUDT_ScalanceSwitchDevice.PNNetworknumber].DeviceStatus[#sUDT_ScalanceSwitchDevice.PNDeviceNumber].DeviceState.Error
	        AND #sx_PowerOk
	        AND NOT #ix_SimulationModeActive
	        AND NOT #sUDT_HMIStatus.Specific.ScalanceSwitchPNSlaveWarning
	    THEN
	        #sUDT_HMIStatus.Specific.ScalanceSwitchPNSlaveError := TRUE;
	    END_IF;

	    // check if Singulator coupler is online
	    IF (NOT "DB_ProfinetDiagnostic".ProfinetNetworks[#sUDT_SingulatorCouplerPNDevice.PNNetworknumber].DeviceStatus[#sUDT_SingulatorCouplerPNDevice.PNDeviceNumber].DeviceState.Exist
	        OR NOT #sUDT_SingulatorCouplerPNDevice.PNDeviceFound)
	        AND #sx_PowerOk
	        AND NOT #ix_SimulationModeActive
	        AND #ix_SingulatorCouplerAvailable
	    THEN
	        #sUDT_HMIStatus.Specific.Singulator_PNSlaveNotOnline := TRUE;
	    END_IF;

	    // Check if Singulator coupler ports are healthy
	    IF #sa_SingulatorPortsStatus[1] XOR #sa_SingulatorPortsStatus[2] THEN
	        #sUDT_HMIStatus.Specific.Singulator_PNSlaveWarning := TRUE;
	    END_IF;

	    // check if Singulator coupler has an error
	    IF "DB_ProfinetDiagnostic".ProfinetNetworks[#sUDT_SingulatorCouplerPNDevice.PNNetworknumber].DeviceStatus[#sUDT_SingulatorCouplerPNDevice.PNDeviceNumber].DeviceState.Error
	        AND #ix_SingulatorCouplerAvailable
	        AND #sx_PowerOk
	        AND NOT #ix_SimulationModeActive
	    THEN
	        #sUDT_HMIStatus.Specific.Singulator_PNSlaveError := TRUE;
	    END_IF;

	    IF NOT #ix_NoFireAlarmActive AND NOT #ix_SimulationModeActive
	    THEN

	        #sUDT_HMIStatus.Specific.FireAlarmActive := TRUE;

	    END_IF;

	    // Unit power supply fault status is set when the input is high

	    IF NOT #ix_UPSOk AND NOT #ix_SimulationModeActive
	    THEN

	        #sUDT_HMIStatus.Specific.UPSSwitchTripped := TRUE;

	    END_IF;

	    IF NOT #ix_24V201T1 AND NOT #ix_SimulationModeActive
	    THEN

	        #sUDT_HMIStatus.Specific.PS_201T1_Tripped := TRUE;

	    END_IF;

	    IF NOT #ix_CBTripped101F4 AND NOT #ix_SimulationModeActive
	    THEN

	        #sUDT_HMIStatus.Specific."230VAC_CB101F4Tripped" := TRUE;

	    END_IF;


	    IF NOT #ix_CBTripped102F1 AND NOT #ix_SimulationModeActive
	    THEN

	        #sUDT_HMIStatus.Specific."230VAC_CB102F1Tripped" := TRUE;

	    END_IF;

	    IF NOT #ix_CBTripped201F1 AND NOT #ix_SimulationModeActive
	    THEN

	        #sUDT_HMIStatus.Specific."24VDC_CB201F1Tripped" := TRUE;

	    END_IF;

	    IF NOT #ix_CBTripped205F5 AND NOT #ix_SimulationModeActive
	    THEN

	        #sUDT_HMIStatus.Specific."24VDC_CB205F5Tripped" := TRUE;

	    END_IF;

	    IF NOT #ix_ScalanceSwitchStatus AND NOT #ix_SimulationModeActive
	    THEN

	        #sUDT_HMIStatus.Specific.ScalanceSwitchStatus := TRUE;
	    END_IF;

	END_REGION

	REGION 9 - Statistics

	    // Unit Power Supply fault statistics

	    IF #sUDT_HMIStatus.Specific.UPSSwitchTripped
	        OR #iqUDT_EquipmentControl.Command.ResetData
	    THEN

	        "FC_Statistics"(ix_Reset := #iqUDT_EquipmentControl.Command.ResetData,
	                        ix_Activate := #sUDT_HMIStatus.Specific.UPSSwitchTripped,
	                        ix_RTrigActivate := #sR_Trig_UPS.Q,
	                        iqUDT_Statistics := #iqUDT_Statistics.UPSFault);

	    END_IF;


	    // 24 VDC Supply fault statistics

	    IF #sUDT_HMIStatus.Specific.FireAlarmActive
	        OR #iqUDT_EquipmentControl.Command.ResetData
	    THEN

	        "FC_Statistics"(ix_Reset := #iqUDT_EquipmentControl.Command.ResetData,
	                        ix_Activate := #sUDT_HMIStatus.Specific.FireAlarmActive,
	                        ix_RTrigActivate := #sR_Trig_FireAlarm.Q,
	                        iqUDT_Statistics := #iqUDT_Statistics.FireAlarm);

	    END_IF;

	    // PN/PN coupler fault statistics

	    IF #sUDT_HMIStatus.Specific."PN_PN_MSP_PNSlaveNotOnline"
	        OR #sUDT_HMIStatus.Specific."PN_PN_MSP_PNSlaveError"
	        OR #iqUDT_EquipmentControl.Command.ResetData
	    THEN

	        "FC_Statistics"(ix_Reset := #iqUDT_EquipmentControl.Command.ResetData,
	                        ix_Activate := #sUDT_HMIStatus.Specific."PN_PN_MSP_PNSlaveNotOnline" OR #sUDT_HMIStatus.Specific."PN_PN_MSP_PNSlaveError",
	                        ix_RTrigActivate := #sR_Trig_PNCoupler.Q,
	                        iqUDT_Statistics := #iqUDT_Statistics."PN/PNCouplerFault");

	    END_IF;

	    // ProSoft coupler fault statistics

	    IF #sUDT_HMIStatus.Specific.Singulator_PNSlaveNotOnline
	        OR #sUDT_HMIStatus.Specific.Singulator_PNSlaveError
	        OR #iqUDT_EquipmentControl.Command.ResetData
	    THEN

	        "FC_Statistics"(ix_Reset := #iqUDT_EquipmentControl.Command.ResetData,
	                        ix_Activate := #sUDT_HMIStatus.Specific.Singulator_PNSlaveNotOnline OR #sUDT_HMIStatus.Specific.Singulator_PNSlaveError,
	                        ix_RTrigActivate := #sR_Trig_ProSoftCoupler.Q,
	                        iqUDT_Statistics := #iqUDT_Statistics.SingulatorCouplerFault);

	    END_IF;

	    // Scalance switch fault statistics

	    IF #sUDT_HMIStatus.Specific.ScalanceSwitchPNSlaveNotOnline
	        OR #sUDT_HMIStatus.Specific.ScalanceSwitchPNSlaveError
	        OR #iqUDT_EquipmentControl.Command.ResetData
	    THEN

	        "FC_Statistics"(ix_Reset := #iqUDT_EquipmentControl.Command.ResetData,
	                        ix_Activate := #sUDT_HMIStatus.Specific.ScalanceSwitchPNSlaveNotOnline OR #sUDT_HMIStatus.Specific.ScalanceSwitchPNSlaveError,
	                        ix_RTrigActivate := #sR_Trig_ScalanceSwitch.Q,
	                        iqUDT_Statistics := #iqUDT_Statistics.ScalanceSwitchFault);

	    END_IF;

	    // Main rack module fault statistics

	    IF #sUDT_HMIStatus.Specific.RackSlotError[0]
	        OR #iqUDT_EquipmentControl.Command.ResetData
	    THEN

	        "FC_Statistics"(ix_Reset := #iqUDT_EquipmentControl.Command.ResetData,
	                        ix_Activate := #sUDT_HMIStatus.Specific.RackSlotError[0],
	                        ix_RTrigActivate := #sR_Trig_MainRackModule.Q,
	                        iqUDT_Statistics := #iqUDT_Statistics.RackModuleFault);

	    END_IF;


	    IF #sUDT_HMIStatus.Specific.PS_201T1_Tripped
	        OR #iqUDT_EquipmentControl.Command.ResetData
	    THEN

	        "FC_Statistics"(ix_Reset := #iqUDT_EquipmentControl.Command.ResetData,
	                        ix_Activate := #sUDT_HMIStatus.Specific.PS_201T1_Tripped,
	                        ix_RTrigActivate := #sR_Trig_24V_201T1.Q,
	                        iqUDT_Statistics := #iqUDT_Statistics.PS_201T1_Tripped);

	    END_IF;

	    IF #sUDT_HMIStatus.Specific."230VAC_CB101F4Tripped"
	        OR #iqUDT_EquipmentControl.Command.ResetData
	    THEN

	        "FC_Statistics"(ix_Reset := #iqUDT_EquipmentControl.Command.ResetData,
	                        ix_Activate := #sUDT_HMIStatus.Specific."230VAC_CB101F4Tripped",
	                        ix_RTrigActivate := #sR_Trig_CB_Tripped_101F4.Q,
	                        iqUDT_Statistics := #iqUDT_Statistics."230VAC_CB101F4Tripped");
	    END_IF;

	    IF #sUDT_HMIStatus.Specific."230VAC_CB102F1Tripped"
	        OR #iqUDT_EquipmentControl.Command.ResetData
	    THEN

	        "FC_Statistics"(ix_Reset := #iqUDT_EquipmentControl.Command.ResetData,
	                        ix_Activate := #sUDT_HMIStatus.Specific."230VAC_CB102F1Tripped",
	                        ix_RTrigActivate := #sR_Trig_CB_Tripped_102F1.Q,
	                        iqUDT_Statistics := #iqUDT_Statistics."230VAC_CB102F1Tripped");
	    END_IF;

	    IF #sUDT_HMIStatus.Specific."24VDC_CB201F1Tripped"
	        OR #iqUDT_EquipmentControl.Command.ResetData
	    THEN

	        "FC_Statistics"(ix_Reset := #iqUDT_EquipmentControl.Command.ResetData,
	                        ix_Activate := #sUDT_HMIStatus.Specific."24VDC_CB201F1Tripped",
	                        ix_RTrigActivate := #sR_Trig_CB_Tripped_201F1.Q,
	                        iqUDT_Statistics := #iqUDT_Statistics."24VDC_CB201F1Tripped");
	    END_IF;

	    IF #sUDT_HMIStatus.Specific."24VDC_CB205F5Tripped"
	        OR #iqUDT_EquipmentControl.Command.ResetData
	    THEN

	        "FC_Statistics"(ix_Reset := #iqUDT_EquipmentControl.Command.ResetData,
	                        ix_Activate := #sUDT_HMIStatus.Specific."24VDC_CB205F5Tripped",
	                        ix_RTrigActivate := #sR_Trig_CB_Tripped_205F5.Q,
	                        iqUDT_Statistics := #iqUDT_Statistics."24VDC_CB205F5Tripped");
	    END_IF;

	    IF #sUDT_HMIStatus.Specific.ScalanceSwitchStatus
	        OR #iqUDT_EquipmentControl.Command.ResetData
	    THEN

	        "FC_Statistics"(ix_Reset := #iqUDT_EquipmentControl.Command.ResetData,
	                        ix_Activate := #sUDT_HMIStatus.Specific.ScalanceSwitchStatus,
	                        ix_RTrigActivate := #sR_Trig_ScalanceSwitchStatus.Q,
	                        iqUDT_Statistics := #iqUDT_Statistics.ScalanceSwitchStatus);
	    END_IF;


	END_REGION

	REGION 10 - Status

	    // Set common error to report
	    #sUDT_CommonStatus.Error := #sUDT_HMIStatus.Specific.PS_201T1_Tripped
	    OR #sUDT_HMIStatus.Specific."230VAC_CB101F4Tripped"
	    OR #sUDT_HMIStatus.Specific."230VAC_CB102F1Tripped"
	    OR #sUDT_HMIStatus.Specific."24VDC_CB201F1Tripped"
	    OR #sUDT_HMIStatus.Specific."24VDC_CB205F5Tripped"
	    OR #sUDT_HMIStatus.Specific.ScalanceSwitchStatus
	    OR #sUDT_HMIStatus.Specific.FireAlarmActive
	    OR #sUDT_HMIStatus.Specific.UPSSwitchTripped
	    OR #sUDT_HMIStatus.Specific."PN_PN_MSP_PNSlaveNotOnline"
	    OR #sUDT_HMIStatus.Specific."PN_PN_MSP_PNSlaveError"
	    OR #sUDT_HMIStatus.Specific.Singulator_PNSlaveNotOnline
	    OR #sUDT_HMIStatus.Specific.Singulator_PNSlaveError
	    OR #sUDT_HMIStatus.Specific.ScalanceSwitchPNSlaveError
	    OR #sUDT_HMIStatus.Specific.ScalanceSwitchPNSlaveNotOnline
	    OR #sUDT_HMIStatus.Specific.IOModule_PNSlaveError
	    OR #sUDT_HMIStatus.Specific.IOModule_PNSlaveNotOnline
	    OR #sUDT_HMIStatus.Specific.RackSlotError[0];

	    // HMI status update
	    IF #sUDT_CommonStatusOld <> #sUDT_CommonStatus                   // update on change
	    THEN

	        // HMI status initialization
	        #sUDT_HMIStatus.Status := 0;


	        // HMI status calculation
	        IF #sUDT_HMIStatus.Specific."PN_PN_MSP_PNSlaveNotOnline"         // Hardware error
	            OR #sUDT_HMIStatus.Specific."PN_PN_MSP_PNSlaveError"
	            OR #sUDT_HMIStatus.Specific.Singulator_PNSlaveNotOnline
	            OR #sUDT_HMIStatus.Specific.Singulator_PNSlaveError
	            OR #sUDT_HMIStatus.Specific.IOModule_PNSlaveError
	            OR #sUDT_HMIStatus.Specific.IOModule_PNSlaveNotOnline
	            OR #sUDT_HMIStatus.Specific.ScalanceSwitchPNSlaveError
	            OR #sUDT_HMIStatus.Specific.ScalanceSwitchPNSlaveNotOnline
	            //  OR #s_UDT_HMIStatus.Specific.RackSlotError[0]
	        THEN

	            #sUDT_HMIStatus.Status := "DB_HMIStatusConfiguration".Error;

	        END_IF;


	        IF #sUDT_HMIStatus.Specific."230VAC_CB101F4Tripped"
	            OR #sUDT_HMIStatus.Specific."230VAC_CB102F1Tripped"
	            OR #sUDT_HMIStatus.Specific."24VDC_CB201F1Tripped"
	            OR #sUDT_HMIStatus.Specific."24VDC_CB205F5Tripped"
	            OR #sUDT_HMIStatus.Specific.PS_201T1_Tripped
	            OR #sUDT_HMIStatus.Specific.UPSSwitchTripped
	        THEN

	            #sUDT_HMIStatus.Status := "DB_HMIStatusConfiguration".CBError;

	        END_IF;

	        IF #sUDT_HMIStatus.Specific.FireAlarmActive                    // Fire alarm
	        THEN

	            #sUDT_HMIStatus.Status := "DB_HMIStatusConfiguration".FireAlarm;

	        END_IF;
	        #sUDT_CommonStatusOld := #sUDT_CommonStatus;                  // Copy status to memory
	        #qUDT_Status := #sUDT_CommonStatus;                           // Copy status to output
	    END_IF;

	    #qUDT_HMIStatus := #sUDT_HMIStatus;                           // Copy HMI status to output

	END_REGION

	REGION 11 - Report to control block

	    // Function to manage report between control block and conveyor block

	    "FC_EquipmentReport"(iUDT_Status := #sUDT_CommonStatus,
	                         iqUDT_Control := #iqUDT_EquipmentControl);

	END_REGION

